C07264=1105.012,382.396,409.215,-179.501,16.996,151.526
C07265=1105.019,382.643,409.178,-179.498,17.001,151.527
C07266=1105.028,383.057,409.117,-179.494,17.008,151.528
C07267=1105.037,383.470,409.056,-179.490,17.016,151.529
C07268=1105.047,383.884,408.995,-179.484,17.024,151.530
C07269=1105.056,384.298,408.934,-179.480,17.032,151.531
C07270=1105.061,384.545,408.897,-179.478,17.037,151.532
C07271=1105.067,384.792,408.860,-179.476,17.041,151.532
C07272=1105.073,385.040,408.823,-179.473,17.046,151.533
C07273=1105.078,385.286,408.787,-179.470,17.051,151.534
C07274=1105.084,385.533,408.750,-179.468,17.056,151.534
C07275=1105.090,385.781,408.713,-179.465,17.060,151.535
C07276=1105.096,386.028,408.677,-179.462,17.065,151.536
C07277=1105.101,386.274,408.640,-179.460,17.070,151.536
C07278=1105.106,386.522,408.603,-179.457,17.075,151.537
C07279=1105.112,386.769,408.566,-179.454,17.080,151.538
C07280=1105.118,387.016,408.529,-179.453,17.084,151.538
C07281=1105.124,387.264,408.492,-179.450,17.089,151.539
C07282=1105.129,387.510,408.456,-179.447,17.094,151.540
C07283=1105.135,387.758,408.419,-179.445,17.098,151.540
C07284=1105.141,388.005,408.382,-179.442,17.104,151.541
C07285=1105.147,388.251,408.344,-179.440,17.108,151.542
C07286=1105.152,388.499,408.307,-179.437,17.113,151.543
C07287=1105.158,388.746,408.270,-179.435,17.118,151.543
C07288=1105.163,388.993,408.234,-179.432,17.123,151.544
C07289=1105.169,389.240,408.197,-179.429,17.128,151.545
C07290=1105.175,389.487,408.160,-179.427,17.133,151.546
C07291=1105.181,389.734,408.122,-179.424,17.138,151.546
C07292=1105.186,389.981,408.085,-179.422,17.143,151.547
C07293=1105.192,390.229,408.048,-179.419,17.148,151.548
C07294=1105.198,390.476,408.012,-179.417,17.153,151.548
C07295=1105.204,390.722,407.974,-179.414,17.158,151.549
C07296=1105.210,390.970,407.937,-179.412,17.164,151.550
C07297=1105.216,391.217,407.900,-179.409,17.168,151.551
C07298=1105.221,391.463,407.863,-179.407,17.174,151.552
C07299=1105.226,391.711,407.826,-179.404,17.179,151.552
C07300=1105.232,391.958,407.789,-179.402,17.184,151.553
C07301=1105.238,392.205,407.751,-179.399,17.189,151.554
C07302=1105.244,392.452,407.714,-179.397,17.194,151.555
C07303=1105.249,392.699,407.676,-179.394,17.199,151.555
C07304=1105.255,392.946,407.639,-179.392,17.204,151.556
C07305=1105.261,393.194,407.602,-179.390,17.210,151.557
C07306=1105.267,393.440,407.564,-179.387,17.215,151.558
C07307=1105.272,393.688,407.527,-179.385,17.220,151.559
C07308=1105.278,393.934,407.489,-179.383,17.225,151.560
C07309=1105.284,394.182,407.452,-179.380,17.231,151.560
C07310=1105.290,394.428,407.415,-179.378,17.236,151.561
C07311=1105.295,394.676,407.378,-179.376,17.241,151.562
C07312=1105.301,394.923,407.340,-179.373,17.247,151.563
C07313=1105.307,395.170,407.303,-179.371,17.252,151.564
C07314=1105.313,395.417,407.265,-179.369,17.257,151.565
C07315=1105.318,395.664,407.228,-179.366,17.263,151.566
C07316=1105.323,395.911,407.190,-179.364,17.268,151.567
C07317=1105.329,396.158,407.152,-179.361,17.274,151.567
C07318=1105.334,396.371,407.119,-179.359,17.278,151.568
C07319=1105.339,396.584,407.087,-179.358,17.283,151.569
C07320=1105.344,396.797,407.055,-179.355,17.288,151.570
C07321=1105.349,397.009,407.023,-179.354,17.293,151.571
C07322=1105.354,397.223,406.990,-179.351,17.298,151.571
C07323=1105.359,397.435,406.958,-179.350,17.302,151.572
C07324=1105.364,397.648,406.925,-179.348,17.307,151.573
C07325=1105.369,397.861,406.892,-179.345,17.312,151.574
C07326=1105.375,398.108,406.855,-179.343,17.317,151.575
C07327=1105.380,398.355,406.818,-179.341,17.323,151.576
C07328=1105.385,398.602,406.779,-179.339,17.328,151.577
C07329=1105.391,398.849,406.741,-179.337,17.334,151.578
C07330=1105.397,399.096,406.704,-179.334,17.340,151.579
C07331=1105.403,399.344,406.666,-179.332,17.346,151.580
C07332=1105.408,399.591,406.628,-179.329,17.351,151.580
C07333=1105.414,399.838,406.590,-179.327,17.357,151.581
C07334=1105.420,400.085,406.552,-179.325,17.363,151.582
C07335=1105.425,400.331,406.514,-179.322,17.369,151.584
C07336=1105.431,400.578,406.476,-179.320,17.375,151.585
C07337=1105.436,400.825,406.438,-179.318,17.380,151.585
C07338=1105.442,401.072,406.400,-179.316,17.386,151.587
C07339=1105.448,401.320,406.362,-179.313,17.392,151.588
C07340=1105.454,401.567,406.324,-179.311,17.398,151.589
C07341=1105.460,401.814,406.287,-179.309,17.404,151.590
C07342=1105.465,402.061,406.248,-179.307,17.409,151.591
C07343=1105.471,402.308,406.211,-179.305,17.416,151.592
C07344=1105.476,402.555,406.172,-179.302,17.422,151.593
C07345=1105.482,402.802,406.134,-179.300,17.428,151.594
C07346=1105.488,403.049,406.096,-179.299,17.434,151.595
C07347=1105.493,403.296,406.058,-179.296,17.440,151.596
C07348=1105.499,403.542,406.019,-179.294,17.446,151.597
C07349=1105.505,403.790,405.981,-179.292,17.452,151.598
C07350=1105.511,404.037,405.942,-179.289,17.458,151.599
C07351=1105.517,404.284,405.905,-179.287,17.464,151.600
C07352=1105.522,404.531,405.866,-179.285,17.470,151.601
C07353=1105.528,404.778,405.828,-179.283,17.476,151.603
C07354=1105.533,405.025,405.790,-179.281,17.482,151.604
C07355=1105.539,405.272,405.752,-179.279,17.488,151.605
C07356=1105.545,405.518,405.713,-179.276,17.495,151.606
C07357=1105.551,405.766,405.675,-179.274,17.501,151.607
C07358=1105.556,406.013,405.637,-179.272,17.508,151.608
C07359=1105.562,406.260,405.598,-179.270,17.514,151.609
C07360=1105.568,406.506,405.560,-179.268,17.520,151.611
C07361=1105.574,406.754,405.521,-179.266,17.527,151.612
C07362=1105.579,407.001,405.483,-179.264,17.532,151.613
C07363=1105.585,407.247,405.444,-179.261,17.539,151.614
C07364=1105.591,407.495,405.406,-179.259,17.545,151.615
C07365=1105.596,407.742,405.367,-179.258,17.552,151.617
C07366=1105.602,407.988,405.329,-179.255,17.558,151.618
C07367=1105.607,408.235,405.290,-179.254,17.565,151.619
C07368=1105.613,408.483,405.252,-179.251,17.572,151.620
C07369=1105.618,408.729,405.213,-179.249,17.578,151.621
C07370=1105.624,408.976,405.174,-179.247,17.584,151.623
C07371=1105.630,409.223,405.135,-179.245,17.591,151.624
C07372=1105.636,409.470,405.097,-179.243,17.598,151.625
C07373=1105.641,409.716,405.058,-179.241,17.604,151.626
C07374=1105.646,409.930,405.025,-179.239,17.610,151.628
C07375=1105.650,410.142,404.992,-179.237,17.616,151.629
C07376=1105.656,410.355,404.958,-179.235,17.622,151.630
C07377=1105.661,410.568,404.924,-179.234,17.627,151.631
C07378=1105.665,410.780,404.891,-179.232,17.633,151.632
C07379=1105.670,410.994,404.857,-179.230,17.639,151.633
C07380=1105.675,411.206,404.824,-179.229,17.645,151.634
C07381=1105.680,411.419,404.791,-179.227,17.651,151.635
C07382=1105.686,411.665,404.752,-179.225,17.657,151.637
C07383=1105.692,411.913,404.713,-179.223,17.664,151.638
C07384=1105.697,412.159,404.674,-179.221,17.671,151.639
C07385=1105.703,412.406,404.635,-179.219,17.678,151.641
C07386=1105.709,412.653,404.596,-179.217,17.685,151.642
C07387=1105.714,412.900,404.557,-179.215,17.692,151.643
C07388=1105.720,413.147,404.518,-179.213,17.699,151.645
C07389=1105.725,413.394,404.480,-179.210,17.706,151.646
C07390=1105.731,413.641,404.440,-179.209,17.713,151.647
C07391=1105.737,413.888,404.401,-179.207,17.720,151.649
C07392=1105.742,414.134,404.362,-179.205,17.726,151.650
C07393=1105.748,414.381,404.323,-179.203,17.734,151.652
C07394=1105.754,414.628,404.285,-179.201,17.741,151.653
C07395=1105.760,414.875,404.245,-179.199,17.748,151.654
C07396=1105.766,415.121,404.206,-179.197,17.755,151.656
C07397=1105.772,415.369,404.167,-179.195,17.762,151.657
C07398=1105.777,415.615,404.128,-179.193,17.770,151.659
C07399=1105.783,415.862,404.088,-179.192,17.776,151.660
C07400=1105.789,416.109,404.049,-179.189,17.784,151.662
C07401=1105.795,416.356,404.010,-179.187,17.791,151.663
C07402=1105.800,416.602,403.971,-179.185,17.799,151.665
C07403=1105.806,416.850,403.931,-179.184,17.805,151.666
C07404=1105.811,417.096,403.892,-179.182,17.813,151.667
C07405=1105.817,417.343,403.852,-179.180,17.820,151.669
C07406=1105.823,417.590,403.813,-179.178,17.828,151.671
C07407=1105.829,417.837,403.774,-179.176,17.835,151.672
C07408=1105.834,418.083,403.735,-179.175,17.843,151.674
C07409=1105.840,418.331,403.695,-179.173,17.850,151.675
C07410=1105.845,418.577,403.656,-179.171,17.858,151.677
C07411=1105.851,418.824,403.616,-179.169,17.865,151.678
C07412=1105.857,419.071,403.577,-179.167,17.873,151.680
C07413=1105.863,419.318,403.538,-179.165,17.881,151.681
C07414=1105.868,419.564,403.497,-179.164,17.888,151.683
C07415=1105.874,419.811,403.458,-179.162,17.895,151.684
C07416=1105.880,420.058,403.419,-179.160,17.903,151.686
C07417=1105.885,420.305,403.379,-179.158,17.911,151.688
C07418=1105.891,420.551,403.339,-179.156,17.919,151.689
C07419=1105.897,420.798,403.300,-179.154,17.927,151.691
C07420=1105.903,421.045,403.260,-179.152,17.934,151.693
C07421=1105.907,421.292,403.221,-179.151,17.942,151.694
C07422=1105.914,421.538,403.180,-179.149,17.950,151.696
C07423=1105.920,421.785,403.141,-179.147,17.958,151.698
C07424=1105.926,422.031,403.101,-179.146,17.965,151.699
C07425=1105.931,422.279,403.061,-179.144,17.973,151.701
C07426=1105.937,422.526,403.022,-179.143,17.982,151.703
C07427=1105.943,422.772,402.982,-179.141,17.989,151.704
C07428=1105.948,423.019,402.942,-179.139,17.997,151.706
C07429=1105.954,423.265,402.902,-179.137,18.005,151.708
C07430=1105.958,423.484,402.867,-179.135,18.013,151.709
C07431=1105.964,423.704,402.832,-179.134,18.020,151.711
C07432=1105.969,423.923,402.795,-179.133,18.027,151.712
C07433=1105.974,424.143,402.760,-179.131,18.035,151.714
C07434=1105.979,424.362,402.725,-179.130,18.042,151.715
C07435=1105.984,424.581,402.689,-179.128,18.050,151.717
C07436=1105.989,424.800,402.654,-179.127,18.057,151.719
C07437=1105.994,425.020,402.619,-179.126,18.064,151.720
C07438=1106.000,425.267,402.578,-179.124,18.072,151.722
C07439=1106.005,425.512,402.538,-179.122,18.080,151.724
C07440=1106.011,425.760,402.498,-179.121,18.088,151.725
C07441=1106.017,426.006,402.458,-179.119,18.098,151.727
C07442=1106.022,426.252,402.418,-179.117,18.106,151.729
C07443=1106.028,426.500,402.378,-179.115,18.114,151.731
C07444=1106.034,426.746,402.337,-179.114,18.123,151.733
C07445=1106.040,426.993,402.297,-179.112,18.131,151.735
C07446=1106.045,427.239,402.257,-179.111,18.139,151.737
C07447=1106.051,427.486,402.217,-179.110,18.148,151.738
C07448=1106.057,427.733,402.177,-179.108,18.156,151.740
C07449=1106.062,427.979,402.136,-179.106,18.165,151.742
C07450=1106.068,428.226,402.096,-179.104,18.174,151.744
C07451=1106.074,428.472,402.056,-179.103,18.183,151.746
C07452=1106.079,428.720,402.015,-179.102,18.191,151.748
C07453=1106.085,428.966,401.976,-179.100,18.200,151.750
C07454=1106.091,429.213,401.935,-179.099,18.209,151.752
C07455=1106.097,429.459,401.894,-179.097,18.218,151.754
C07456=1106.103,429.706,401.854,-179.096,18.226,151.756
C07457=1106.108,429.952,401.814,-179.094,18.235,151.758
C07458=1106.114,430.199,401.773,-179.093,18.244,151.760
C07459=1106.120,430.445,401.733,-179.091,18.254,151.762
C07460=1106.125,430.691,401.692,-179.090,18.262,151.764
C07461=1106.131,430.938,401.652,-179.089,18.271,151.766
C07462=1106.136,431.185,401.611,-179.088,18.280,151.768
C07463=1106.142,431.432,401.570,-179.086,18.290,151.770
C07464=1106.148,431.678,401.530,-179.084,18.298,151.772
C07465=1106.153,431.925,401.490,-179.083,18.308,151.774
C07466=1106.159,432.171,401.449,-179.081,18.317,151.776
C07467=1106.165,432.418,401.407,-179.080,18.326,151.778
C07468=1106.171,432.664,401.367,-179.079,18.335,151.780
C07469=1106.177,432.911,401.327,-179.077,18.345,151.782
C07470=1106.182,433.157,401.286,-179.076,18.354,151.784
C07471=1106.188,433.404,401.245,-179.075,18.363,151.787
C07472=1106.194,433.650,401.204,-179.073,18.373,151.789
C07473=1106.199,433.897,401.163,-179.072,18.382,151.791
C07474=1106.205,434.144,401.123,-179.071,18.391,151.793
C07475=1106.210,434.390,401.082,-179.070,18.401,151.795
C07476=1106.216,434.636,401.041,-179.069,18.410,151.797
C07477=1106.222,434.883,401.000,-179.067,18.421,151.800
C07478=1106.227,435.130,400.959,-179.066,18.430,151.802
C07479=1106.233,435.376,400.918,-179.065,18.439,151.804
C07480=1106.238,435.622,400.877,-179.064,18.449,151.806
C07481=1106.244,435.868,400.836,-179.063,18.459,151.809
C07482=1106.250,436.115,400.795,-179.061,18.469,151.811
C07483=1106.255,436.362,400.754,-179.060,18.478,151.813
C07484=1106.261,436.608,400.713,-179.059,18.488,151.815
C07485=1106.267,436.855,400.672,-179.058,18.498,151.818
C07486=1106.272,437.072,400.636,-179.057,18.507,151.820
C07487=1106.277,437.290,400.600,-179.056,18.516,151.822
C07488=1106.282,437.508,400.563,-179.055,18.524,151.824
C07489=1106.287,437.726,400.526,-179.054,18.533,151.826
C07490=1106.292,437.944,400.490,-179.053,18.542,151.828
C07491=1106.297,438.162,400.454,-179.052,18.551,151.830
C07492=1106.302,438.380,400.418,-179.051,18.560,151.832
C07493=1106.307,438.598,400.381,-179.050,18.569,151.834
C07494=1106.313,438.844,400.340,-179.049,18.579,151.837
C07495=1106.318,439.091,400.299,-179.048,18.589,151.839
C07496=1106.324,439.337,400.257,-179.047,18.600,151.842
C07497=1106.330,439.583,400.216,-179.046,18.609,151.844
C07498=1106.336,439.829,400.175,-179.045,18.620,151.846
C07499=1106.341,440.076,400.133,-179.044,18.630,151.849
C07500=1106.347,440.323,400.092,-179.043,18.641,151.851
C07501=1106.353,440.569,400.050,-179.041,18.651,151.854
C07502=1106.359,440.815,400.009,-179.041,18.661,151.856
C07503=1106.365,441.062,399.968,-179.040,18.672,151.859
C07504=1106.370,441.308,399.926,-179.039,18.682,151.861
C07505=1106.376,441.555,399.885,-179.038,18.693,151.864
C07506=1106.382,441.801,399.843,-179.037,18.704,151.866
C07507=1106.388,442.047,399.802,-179.037,18.714,151.869
C07508=1106.393,442.293,399.760,-179.036,18.725,151.872
C07509=1106.399,442.540,399.718,-179.034,18.736,151.874
C07510=1106.405,442.786,399.677,-179.034,18.747,151.877
C07511=1106.410,443.032,399.635,-179.033,18.758,151.879
C07512=1106.416,443.279,399.593,-179.032,18.769,151.882
C07513=1106.421,443.525,399.551,-179.032,18.779,151.885
C07514=1106.427,443.771,399.510,-179.031,18.790,151.887
C07515=1106.433,444.018,399.468,-179.030,18.801,151.890
C07516=1106.438,444.264,399.426,-179.030,18.812,151.893
C07517=1106.444,444.510,399.385,-179.029,18.823,151.895
C07518=1106.449,444.757,399.343,-179.029,18.834,151.898
C07519=1106.455,445.003,399.301,-179.029,18.845,151.901
C07520=1106.461,445.249,399.259,-179.030,18.855,151.904
C07521=1106.467,445.496,399.218,-179.030,18.866,151.907
C07522=1106.472,445.742,399.176,-179.030,18.877,151.909
C07523=1106.478,445.988,399.134,-179.031,18.887,151.912
C07524=1106.483,446.234,399.091,-179.032,18.898,151.915
C07525=1106.489,446.480,399.050,-179.032,18.909,151.918
C07526=1106.494,446.727,399.008,-179.033,18.920,151.921
C07527=1106.501,446.974,398.966,-179.034,18.930,151.924
C07528=1106.506,447.220,398.924,-179.035,18.941,151.927
C07529=1106.512,447.467,398.883,-179.036,18.952,151.930
C07530=1106.518,447.713,398.840,-179.037,18.963,151.933
C07531=1106.523,447.959,398.798,-179.039,18.973,151.936
C07532=1106.529,448.205,398.756,-179.040,18.984,151.939
C07533=1106.534,448.452,398.714,-179.042,18.994,151.942
C07534=1106.539,448.698,398.671,-179.043,19.005,151.945
C07535=1106.546,448.945,398.630,-179.045,19.015,151.948
C07536=1106.551,449.191,398.588,-179.047,19.026,151.951
C07537=1106.558,449.437,398.545,-179.049,19.037,151.954
C07538=1106.563,449.683,398.503,-179.050,19.047,151.957
C07539=1106.568,449.930,398.461,-179.053,19.058,151.960
C07540=1106.574,450.175,398.419,-179.054,19.068,151.963
C07541=1106.579,450.422,398.377,-179.057,19.079,151.966
C07542=1106.174,450.414,398.257,-179.136,19.309,152.039
C07543=1106.168,450.169,398.299,-179.134,19.299,152.036
C07544=1106.162,449.922,398.341,-179.132,19.288,152.033
C07545=1106.157,449.676,398.384,-179.130,19.277,152.030
C07546=1106.151,449.430,398.425,-179.128,19.267,152.027
C07547=1106.145,449.183,398.468,-179.126,19.256,152.024
C07548=1106.140,448.937,398.510,-179.125,19.245,152.021
C07549=1106.134,448.691,398.552,-179.123,19.235,152.018
C07550=1106.129,448.444,398.594,-179.121,19.224,152.015
C07551=1106.123,448.198,398.637,-179.120,19.213,152.012
C07552=1106.116,447.952,398.678,-179.118,19.203,152.009
C07553=1106.111,447.705,398.720,-179.117,19.192,152.006
C07554=1106.105,447.459,398.763,-179.116,19.181,152.003
C07555=1106.100,447.213,398.805,-179.115,19.170,152.000
C07556=1106.095,446.966,398.847,-179.114,19.160,151.997
C07557=1106.089,446.720,398.888,-179.113,19.149,151.994
C07558=1106.083,446.474,398.931,-179.112,19.138,151.991
C07559=1106.077,446.228,398.972,-179.112,19.127,151.988
C07560=1106.071,445.981,399.015,-179.112,19.116,151.986
C07561=1106.066,445.734,399.057,-179.111,19.106,151.983
C07562=1106.060,445.489,399.099,-179.111,19.095,151.980
C07563=1106.055,445.242,399.141,-179.110,19.084,151.977
C07564=1106.049,444.996,399.183,-179.110,19.073,151.974
C07565=1106.043,444.750,399.224,-179.110,19.062,151.971
C07566=1106.038,444.503,399.266,-179.110,19.051,151.969
C07567=1106.032,444.257,399.308,-179.110,19.040,151.966
C07568=1106.026,444.011,399.350,-179.111,19.029,151.963
C07569=1106.020,443.765,399.392,-179.112,19.018,151.960
C07570=1106.015,443.519,399.434,-179.112,19.008,151.958
C07571=1106.009,443.272,399.475,-179.113,18.996,151.955
C07572=1106.004,443.026,399.517,-179.114,18.985,151.952
C07573=1105.998,442.780,399.559,-179.115,18.974,151.950
C07574=1105.992,442.533,399.600,-179.115,18.964,151.947
C07575=1105.987,442.287,399.642,-179.117,18.953,151.945
C07576=1105.980,442.040,399.684,-179.118,18.942,151.942
C07577=1105.975,441.795,399.725,-179.118,18.931,151.939
C07578=1105.969,441.548,399.767,-179.119,18.920,151.937
C07579=1105.964,441.301,399.808,-179.121,18.909,151.934
C07580=1105.958,441.055,399.849,-179.121,18.899,151.932
C07581=1105.952,440.809,399.891,-179.122,18.888,151.929
C07582=1105.947,440.562,399.933,-179.123,18.878,151.927
C07583=1105.941,440.316,399.974,-179.124,18.867,151.924
C07584=1105.935,440.070,400.016,-179.126,18.857,151.922
C07585=1105.929,439.824,400.057,-179.126,18.847,151.919
C07586=1105.923,439.577,400.098,-179.127,18.836,151.917
C07587=1105.917,439.331,400.140,-179.128,18.826,151.914
C07588=1105.912,439.084,400.182,-179.130,18.815,151.912
C07589=1105.906,438.838,400.223,-179.131,18.805,151.910
C07590=1105.901,438.591,400.264,-179.132,18.795,151.907
C07591=1105.896,438.375,400.300,-179.133,18.786,151.905
C07592=1105.890,438.159,400.336,-179.134,18.777,151.903
C07593=1105.885,437.943,400.373,-179.135,18.768,151.901
C07594=1105.880,437.727,400.409,-179.136,18.759,151.899
C07595=1105.875,437.512,400.444,-179.137,18.750,151.897
C07596=1105.870,437.297,400.480,-179.138,18.742,151.895
C07597=1105.865,437.081,400.517,-179.139,18.733,151.893
C07598=1105.860,436.865,400.553,-179.140,18.724,151.891
C07599=1105.854,436.618,400.594,-179.141,18.714,151.888
C07600=1105.848,436.372,400.635,-179.143,18.704,151.886
C07601=1105.843,436.126,400.675,-179.143,18.695,151.884
C07602=1105.837,435.879,400.717,-179.145,18.684,151.881
C07603=1105.832,435.633,400.758,-179.146,18.675,151.879
C07604=1105.826,435.386,400.799,-179.148,18.665,151.877
C07605=1105.820,435.140,400.840,-179.149,18.655,151.875
C07606=1105.814,434.893,400.881,-179.150,18.646,151.872
C07607=1105.809,434.647,400.922,-179.151,18.636,151.870
C07608=1105.804,434.400,400.962,-179.152,18.626,151.868
C07609=1105.798,434.154,401.004,-179.154,18.616,151.866
C07610=1105.792,433.907,401.045,-179.155,18.607,151.864
C07611=1105.786,433.661,401.085,-179.157,18.597,151.861
C07612=1105.780,433.414,401.127,-179.158,18.588,151.859
C07613=1105.775,433.168,401.167,-179.159,18.579,151.857
C07614=1105.770,432.921,401.208,-179.161,18.569,151.855
C07615=1105.764,432.675,401.249,-179.162,18.560,151.853
C07616=1105.758,432.428,401.290,-179.163,18.550,151.851
C07617=1105.752,432.182,401.330,-179.165,18.541,151.849
C07618=1105.747,431.936,401.371,-179.166,18.532,151.847
C07619=1105.741,431.689,401.411,-179.167,18.523,151.845
C07620=1105.735,431.442,401.452,-179.169,18.513,151.842
C07621=1105.730,431.195,401.493,-179.171,18.504,151.840
C07622=1105.723,430.949,401.534,-179.172,18.495,151.838
C07623=1105.718,430.703,401.574,-179.173,18.486,151.836
C07624=1105.712,430.456,401.615,-179.175,18.477,151.834
C07625=1105.707,430.210,401.656,-179.176,18.468,151.832
C07626=1105.701,429.963,401.696,-179.178,18.459,151.830
C07627=1105.695,429.717,401.736,-179.179,18.450,151.828
C07628=1105.690,429.470,401.777,-179.181,18.441,151.826
C07629=1105.684,429.223,401.818,-179.182,18.432,151.824
C07630=1105.678,428.977,401.858,-179.183,18.423,151.822
C07631=1105.672,428.730,401.898,-179.185,18.415,151.820
C07632=1105.667,428.484,401.939,-179.187,18.405,151.818
C07633=1105.661,428.237,401.978,-179.189,18.397,151.816
C07634=1105.655,427.990,402.019,-179.190,18.388,151.814
C07635=1105.649,427.743,402.059,-179.191,18.380,151.813
C07636=1105.644,427.497,402.100,-179.193,18.371,151.811
C07637=1105.638,427.250,402.140,-179.195,18.363,151.809
C07638=1105.632,427.004,402.180,-179.197,18.353,151.807
C07639=1105.627,426.757,402.220,-179.198,18.345,151.805
C07640=1105.621,426.511,402.260,-179.200,18.336,151.803
C07641=1105.615,426.264,402.301,-179.201,18.328,151.801
C07642=1105.609,426.017,402.341,-179.203,18.319,151.800
C07643=1105.604,425.771,402.381,-179.204,18.311,151.798
C07644=1105.598,425.524,402.422,-179.206,18.303,151.796
C07645=1105.592,425.277,402.462,-179.207,18.294,151.794
C07646=1105.587,425.031,402.501,-179.209,18.286,151.792
C07647=1105.581,424.811,402.537,-179.211,18.278,151.791
C07648=1105.576,424.592,402.573,-179.212,18.271,151.789
C07649=1105.572,424.372,402.608,-179.214,18.264,151.788
C07650=1105.567,424.153,402.644,-179.215,18.256,151.786
C07651=1105.561,423.933,402.679,-179.216,18.249,151.784
C07652=1105.556,423.714,402.715,-179.219,18.241,151.783
C07653=1105.552,423.494,402.750,-179.220,18.234,151.781
C07654=1105.547,423.275,402.786,-179.222,18.227,151.780
C07655=1105.541,423.028,402.826,-179.224,18.219,151.778
C07656=1105.534,422.782,402.866,-179.225,18.211,151.776
C07657=1105.530,422.535,402.906,-179.227,18.202,151.775
C07658=1105.523,422.288,402.946,-179.229,18.194,151.773
C07659=1105.517,422.041,402.985,-179.230,18.187,151.771
C07660=1105.512,421.795,403.025,-179.232,18.179,151.770
C07661=1105.506,421.548,403.065,-179.233,18.171,151.768
C07662=1105.500,421.301,403.105,-179.235,18.163,151.766
C07663=1105.495,421.054,403.144,-179.237,18.155,151.765
C07664=1105.489,420.808,403.184,-179.239,18.147,151.763
C07665=1105.483,420.561,403.223,-179.241,18.140,151.761
C07666=1105.477,420.314,403.263,-179.243,18.132,151.760
C07667=1105.472,420.067,403.304,-179.245,18.124,151.758
C07668=1105.466,419.821,403.343,-179.247,18.116,151.756
C07669=1105.460,419.574,403.382,-179.248,18.108,151.755
C07670=1105.455,419.327,403.421,-179.250,18.100,151.753
C07671=1105.449,419.080,403.462,-179.252,18.093,151.752
C07672=1105.444,418.834,403.501,-179.254,18.086,151.750
C07673=1105.438,418.587,403.540,-179.256,18.078,151.749
C07674=1105.432,418.340,403.579,-179.258,18.070,151.747
C07675=1105.427,418.093,403.619,-179.260,18.062,151.745
C07676=1105.421,417.847,403.659,-179.262,18.055,151.744
C07677=1105.415,417.599,403.698,-179.263,18.047,151.742
C07678=1105.409,417.354,403.738,-179.265,18.040,151.741
C07679=1105.403,417.106,403.777,-179.267,18.033,151.739
C07680=1105.399,416.860,403.817,-179.269,18.025,151.738
C07681=1105.392,416.613,403.856,-179.271,18.017,151.736
C07682=1105.387,416.366,403.895,-179.273,18.010,151.735
C07683=1105.381,416.119,403.935,-179.275,18.003,151.733
C07684=1105.375,415.872,403.974,-179.277,17.996,151.732
C07685=1105.369,415.625,404.013,-179.279,17.988,151.730
C07686=1105.363,415.378,404.053,-179.281,17.981,151.729
C07687=1105.358,415.131,404.091,-179.282,17.974,151.728
C07688=1105.352,414.884,404.130,-179.285,17.967,151.726
C07689=1105.347,414.638,404.170,-179.287,17.960,151.725
C07690=1105.341,414.391,404.209,-179.288,17.953,151.723
C07691=1105.335,414.144,404.248,-179.291,17.946,151.722
C07692=1105.330,413.898,404.287,-179.293,17.938,151.720
C07693=1105.324,413.651,404.327,-179.294,17.932,151.719
C07694=1105.318,413.403,404.365,-179.296,17.924,151.718
C07695=1105.312,413.157,404.404,-179.299,17.917,151.716
C07696=1105.306,412.910,404.443,-179.300,17.910,151.715
C07697=1105.300,412.663,404.482,-179.303,17.903,151.714
C07698=1105.295,412.416,404.521,-179.305,17.896,151.712
C07699=1105.289,412.169,404.560,-179.306,17.889,151.711
C07700=1105.283,411.922,404.599,-179.309,17.882,151.709
C07701=1105.278,411.675,404.637,-179.311,17.875,151.708
C07702=1105.272,411.428,404.677,-179.313,17.869,151.707
C07703=1105.267,411.215,404.710,-179.314,17.862,151.706
C07704=1105.262,411.003,404.744,-179.316,17.857,151.704
C07705=1105.257,410.790,404.777,-179.318,17.851,151.703
C07706=1105.252,410.577,404.811,-179.319,17.845,151.702
C07707=1105.248,410.365,404.845,-179.321,17.839,151.701
C07708=1105.243,410.151,404.877,-179.323,17.833,151.700
C07709=1105.238,409.938,404.911,-179.325,17.828,151.699
C07710=1105.233,409.725,404.945,-179.327,17.821,151.698
C07711=1105.227,409.479,404.984,-179.329,17.815,151.696
C07712=1105.222,409.232,405.022,-179.331,17.808,151.695
C07713=1105.216,408.984,405.061,-179.333,17.802,151.694
C07714=1105.210,408.738,405.099,-179.335,17.795,151.693
C07715=1105.205,408.491,405.138,-179.337,17.788,151.691
C07716=1105.199,408.244,405.177,-179.339,17.781,151.690
C07717=1105.194,407.996,405.215,-179.341,17.776,151.689
C07718=1105.187,407.750,405.254,-179.344,17.769,151.688
C07719=1105.182,407.503,405.292,-179.346,17.762,151.686
C07720=1105.177,407.256,405.331,-179.348,17.755,151.685
C07721=1105.170,407.009,405.369,-179.350,17.749,151.684
C07722=1105.165,406.762,405.408,-179.352,17.743,151.683
C07723=1105.159,406.515,405.447,-179.354,17.737,151.682
C07724=1105.154,406.268,405.486,-179.356,17.730,151.680
C07725=1105.148,406.021,405.523,-179.359,17.724,151.679
C07726=1105.142,405.774,405.562,-179.360,17.717,151.678
C07727=1105.136,405.527,405.600,-179.362,17.711,151.677
C07728=1105.131,405.280,405.639,-179.365,17.705,151.676
C07729=1105.126,405.033,405.677,-179.367,17.699,151.675
C07730=1105.119,404.786,405.715,-179.369,17.692,151.674
C07731=1105.114,404.539,405.754,-179.371,17.686,151.672
C07732=1105.108,404.292,405.791,-179.373,17.680,151.671
C07733=1105.103,404.046,405.831,-179.376,17.674,151.670
C07734=1105.096,403.798,405.869,-179.378,17.668,151.669
C07735=1105.091,403.551,405.907,-179.380,17.662,151.668
C07736=1105.085,403.305,405.945,-179.383,17.655,151.667
C07737=1105.080,403.057,405.983,-179.385,17.650,151.666
C07738=1105.073,402.810,406.021,-179.387,17.644,151.665
C07739=1105.068,402.563,406.060,-179.389,17.637,151.664
C07740=1105.062,402.316,406.097,-179.391,17.631,151.663
C07741=1105.057,402.069,406.136,-179.393,17.625,151.661
C07742=1105.051,401.822,406.173,-179.395,17.620,151.661
C07743=1105.045,401.575,406.212,-179.398,17.613,151.659
C07744=1105.040,401.328,406.250,-179.400,17.608,151.658
C07745=1105.034,401.081,406.288,-179.402,17.602,151.657
C07746=1105.029,400.834,406.326,-179.404,17.596,151.656
C07747=1105.023,400.587,406.364,-179.407,17.589,151.655
C07748=1105.017,400.340,406.402,-179.409,17.584,151.654
C07749=1105.011,400.093,406.440,-179.411,17.578,151.653
C07750=1105.005,399.846,406.478,-179.414,17.572,151.652
C07751=1105.000,399.599,406.516,-179.416,17.566,151.651
C07752=1104.994,399.352,406.553,-179.418,17.560,151.650
C07753=1104.988,399.105,406.591,-179.421,17.555,151.649
C07754=1104.983,398.858,406.629,-179.423,17.549,151.648
C07755=1104.977,398.611,406.667,-179.425,17.544,151.647
C07756=1104.971,398.364,406.705,-179.428,17.537,151.646
C07757=1104.965,398.116,406.742,-179.430,17.532,151.645
C07758=1104.960,397.869,406.781,-179.432,17.526,151.644
C07759=1104.955,397.657,406.813,-179.434,17.522,151.644
C07760=1104.950,397.443,406.846,-179.436,17.516,151.643
C07761=1104.945,397.231,406.879,-179.438,17.512,151.642
C07762=1104.940,397.017,406.911,-179.440,17.507,151.641
C07763=1104.936,396.805,406.944,-179.442,17.502,151.640
C07764=1104.931,396.591,406.976,-179.445,17.497,151.639
C07765=1104.925,396.379,407.008,-179.446,17.492,151.639
C07766=1104.921,396.166,407.040,-179.448,17.488,151.638
C07767=1104.915,395.919,407.079,-179.451,17.482,151.637
C07768=1104.910,395.672,407.116,-179.453,17.477,151.636
C07769=1104.903,395.424,407.154,-179.455,17.471,151.635
C07770=1104.898,395.177,407.191,-179.458,17.466,151.634
C07771=1104.892,394.930,407.229,-179.460,17.460,151.633
C07772=1104.886,394.683,407.266,-179.463,17.455,151.633
C07773=1104.880,394.436,407.303,-179.465,17.450,151.632
C07774=1104.874,394.189,407.341,-179.467,17.444,151.631
C07775=1104.869,393.942,407.378,-179.469,17.439,151.630
C07776=1104.864,393.695,407.416,-179.472,17.434,151.629
C07777=1104.858,393.447,407.453,-179.474,17.428,151.628
C07778=1104.852,393.201,407.491,-179.476,17.423,151.627
C07779=1104.847,392.953,407.528,-179.479,17.418,151.627
C07780=1104.841,392.706,407.565,-179.481,17.413,151.626
C07781=1104.836,392.460,407.603,-179.485,17.407,151.625
C07782=1104.830,392.213,407.640,-179.487,17.402,151.624
C07783=1104.824,391.966,407.678,-179.490,17.396,151.623
C07784=1104.819,391.718,407.715,-179.492,17.391,151.623
C07785=1104.812,391.471,407.751,-179.494,17.386,151.622
C07786=1104.806,391.225,407.789,-179.497,17.381,151.621
C07787=1104.801,390.977,407.826,-179.499,17.376,151.620
C07788=1104.795,390.730,407.863,-179.502,17.371,151.619
C07789=1104.789,390.483,407.901,-179.504,17.365,151.619
C07790=1104.784,390.236,407.938,-179.507,17.361,151.618
C07791=1104.778,389.988,407.975,-179.509,17.355,151.617
C07792=1104.772,389.741,408.011,-179.512,17.350,151.616
C07793=1104.766,389.495,408.049,-179.515,17.346,151.616
C07794=1104.760,389.247,408.086,-179.517,17.340,151.615
C07795=1104.755,389.000,408.123,-179.519,17.335,151.614
C07796=1104.750,388.753,408.160,-179.522,17.330,151.613
C07797=1104.744,388.507,408.197,-179.525,17.325,151.613
C07798=1104.737,388.260,408.234,-179.527,17.321,151.612
C07799=1104.732,388.012,408.271,-179.529,17.316,151.611
C07800=1104.726,387.765,408.308,-179.532,17.311,151.610
C07801=1104.721,387.517,408.345,-179.534,17.306,151.610
C07802=1104.715,387.271,408.381,-179.537,17.301,151.609
C07803=1104.709,387.024,408.418,-179.539,17.296,151.608
C07804=1104.704,386.776,408.455,-179.542,17.291,151.608
C07805=1104.698,386.529,408.492,-179.545,17.286,151.607
C07806=1104.691,386.283,408.529,-179.547,17.281,151.606
C07807=1104.686,386.036,408.566,-179.550,17.276,151.605
C07808=1104.681,385.789,408.603,-179.553,17.272,151.605
C07809=1104.675,385.541,408.640,-179.555,17.267,151.604
C07810=1104.669,385.294,408.676,-179.558,17.262,151.603
C07811=1104.664,385.046,408.713,-179.560,17.257,151.603
C07812=1104.659,384.799,408.749,-179.562,17.253,151.602
C07813=1104.652,384.552,408.786,-179.565,17.248,151.601
C07814=1104.647,384.305,408.823,-179.568,17.243,151.601
C07815=1104.637,383.891,408.884,-179.572,17.235,151.600
C07816=1104.629,383.477,408.946,-179.577,17.227,151.599
C07817=1104.619,383.063,409.007,-179.581,17.219,151.598
C07818=1104.609,382.651,409.069,-179.586,17.212,151.597
C07819=1104.603,382.403,409.104,-179.589,17.207,151.596
C07820=1104.598,382.155,409.141,-179.591,17.202,151.595
C07821=1104.591,381.908,409.178,-179.593,17.198,151.595
C07822=1104.586,381.661,409.215,-179.596,17.194,151.594
C07823=1104.580,381.414,409.250,-179.599,17.189,151.594
C07824=1104.575,381.167,409.287,-179.602,17.184,151.593
C07825=1104.568,380.920,409.324,-179.605,17.180,151.592
C07826=1104.564,380.672,409.360,-179.607,17.176,151.592
C07827=1104.557,380.425,409.396,-179.609,17.171,151.591
C07828=1104.551,380.178,409.433,-179.612,17.167,151.591
C07829=1104.546,379.930,409.469,-179.615,17.162,151.590
C07830=1104.540,379.684,409.505,-179.618,17.158,151.590
C07831=1104.534,379.437,409.542,-179.620,17.153,151.589
C07832=1104.528,379.189,409.578,-179.623,17.149,151.589
C07833=1104.523,378.942,409.614,-179.626,17.145,151.588
C07834=1104.517,378.695,409.650,-179.629,17.140,151.587
C07835=1104.511,378.447,409.687,-179.631,17.136,151.587
C07836=1104.506,378.200,409.723,-179.634,17.132,151.586
C07837=1104.500,377.953,409.759,-179.637,17.127,151.586
C07838=1104.495,377.706,409.795,-179.640,17.122,151.585
C07839=1104.489,377.459,409.831,-179.642,17.119,151.585
C07840=1104.483,377.211,409.867,-179.645,17.114,151.584
C07841=1104.478,376.964,409.904,-179.648,17.110,151.584
C07842=1104.472,376.717,409.940,-179.651,17.105,151.583
C07843=1104.466,376.469,409.975,-179.653,17.101,151.583
C07844=1104.461,376.222,410.012,-179.656,17.097,151.582
C07845=1104.455,375.975,410.048,-179.659,17.093,151.582
C07846=1104.449,375.728,410.084,-179.661,17.089,151.581
C07847=1104.444,375.480,410.120,-179.664,17.084,151.581
C07848=1104.438,375.233,410.155,-179.667,17.080,151.580
C07849=1104.432,374.986,410.191,-179.670,17.076,151.580
C07850=1104.427,374.738,410.228,-179.672,17.072,151.579
C07851=1104.421,374.491,410.264,-179.675,17.067,151.579
C07852=1104.415,374.244,410.299,-179.678,17.063,151.578
C07853=1104.410,373.997,410.335,-179.681,17.060,151.578
C07854=1104.404,373.750,410.371,-179.684,17.055,151.578
C07855=1104.398,373.502,410.407,-179.687,17.051,151.577
C07856=1104.393,373.255,410.443,-179.689,17.047,151.577
C07857=1104.387,373.007,410.479,-179.692,17.043,151.576
C07858=1104.381,372.761,410.515,-179.695,17.039,151.576
C07859=1104.375,372.513,410.550,-179.697,17.035,151.575
C07860=1104.370,372.266,410.586,-179.700,17.031,151.575
C07861=1104.364,372.018,410.621,-179.704,17.027,151.575
C07862=1104.358,371.771,410.657,-179.706,17.023,151.574
C07863=1104.353,371.524,410.693,-179.709,17.019,151.574
C07864=1104.347,371.276,410.729,-179.711,17.015,151.573
C07865=1104.341,371.029,410.764,-179.715,17.011,151.573
C07866=1104.335,370.781,410.800,-179.718,17.007,151.573
C07867=1104.327,370.394,410.856,-179.722,17.001,151.572
C07868=1104.317,370.008,410.911,-179.726,16.995,151.571
C07869=1104.309,369.621,410.966,-179.731,16.989,151.571
C07870=1104.300,369.234,411.022,-179.736,16.983,151.570
C07871=1104.294,368.986,411.058,-179.738,16.979,151.570
C07872=1104.289,368.739,411.094,-179.741,16.975,151.569
C07873=1104.283,368.491,411.129,-179.744,16.972,151.569
C07874=1104.277,368.244,411.165,-179.747,16.968,151.569
C07875=1104.271,367.997,411.200,-179.750,16.964,151.568
C07876=1104.266,367.749,411.235,-179.753,16.960,151.568
C07877=1104.260,367.502,411.271,-179.756,16.956,151.568
C07878=1104.255,367.255,411.306,-179.758,16.952,151.567
C07879=1104.249,367.008,411.341,-179.762,16.948,151.567
C07880=1104.243,366.760,411.377,-179.764,16.945,151.567
C07881=1104.238,366.512,411.412,-179.767,16.941,151.566
C07882=1104.232,366.265,411.448,-179.771,16.937,151.566
C07883=1104.226,366.018,411.482,-179.773,16.934,151.566
C07884=1104.220,365.770,411.518,-179.776,16.930,151.565
C07885=1104.215,365.523,411.553,-179.779,16.926,151.565
C07886=1104.209,365.276,411.588,-179.782,16.922,151.565
C07887=1104.203,365.028,411.624,-179.785,16.919,151.564
C07888=1104.198,364.780,411.658,-179.788,16.915,151.564
C07889=1104.192,364.533,411.694,-179.791,16.912,151.564
C07890=1104.186,364.286,411.729,-179.794,16.908,151.564
C07891=1104.181,364.039,411.764,-179.796,16.905,151.563
C07892=1104.175,363.791,411.799,-179.800,16.901,151.563
C07893=1104.170,363.543,411.834,-179.802,16.898,151.563
C07894=1104.163,363.296,411.869,-179.806,16.894,151.562
C07895=1104.158,363.048,411.904,-179.808,16.890,151.562
C07896=1104.152,362.801,411.939,-179.812,16.887,151.562
C07897=1104.147,362.553,411.974,-179.814,16.883,151.562
C07898=1104.141,362.306,412.009,-179.817,16.879,151.561
C07899=1104.135,362.058,412.044,-179.820,16.876,151.561
C07900=1104.129,361.811,412.079,-179.823,16.872,151.561
C07901=1104.124,361.564,412.114,-179.826,16.869,151.561
C07902=1104.118,361.316,412.149,-179.829,16.865,151.560
C07903=1104.112,361.069,412.184,-179.832,16.862,151.560
C07904=1104.107,360.822,412.219,-179.835,16.858,151.560
C07905=1104.101,360.574,412.254,-179.838,16.855,151.560
C07906=1104.095,360.326,412.288,-179.841,16.851,151.559
C07907=1104.090,360.079,412.324,-179.844,16.848,151.559
C07908=1104.084,359.831,412.358,-179.847,16.845,151.559
C07909=1104.078,359.583,412.393,-179.850,16.841,151.559
C07910=1104.072,359.337,412.427,-179.853,16.838,151.558
C07911=1104.067,359.089,412.462,-179.857,16.835,151.558
C07912=1104.061,358.841,412.497,-179.859,16.831,151.558
C07913=1104.055,358.594,412.532,-179.863,16.828,151.558
C07914=1104.050,358.347,412.566,-179.865,16.825,151.558
C07915=1104.044,358.099,412.601,-179.869,16.821,151.558
C07916=1104.039,357.851,412.635,-179.871,16.818,151.557
C07917=1104.032,357.604,412.670,-179.874,16.815,151.557
C07918=1104.027,357.356,412.705,-179.878,16.811,151.557
C07919=1104.018,356.984,412.757,-179.882,16.806,151.557
C07920=1104.010,356.612,412.809,-179.887,16.802,151.556
C07921=1104.001,356.240,412.861,-179.892,16.796,151.556
C07922=1103.992,355.868,412.913,-179.896,16.792,151.556
C07923=1103.987,355.620,412.947,-179.899,16.788,151.556
C07924=1103.981,355.373,412.981,-179.902,16.785,151.555
C07925=1103.976,355.125,413.016,-179.905,16.782,151.555
C07926=1103.970,354.877,413.050,-179.908,16.778,151.555
C07927=1103.965,354.630,413.085,-179.911,16.775,151.555
C07928=1103.959,354.382,413.119,-179.915,16.772,151.555
C07929=1103.953,354.135,413.153,-179.917,16.769,151.555
C07930=1103.948,353.887,413.188,-179.920,16.766,151.555
C07931=1103.941,353.639,413.222,-179.924,16.763,151.554
C07932=1103.936,353.392,413.257,-179.927,16.760,151.554
C07933=1103.930,353.145,413.291,-179.929,16.757,151.554
C07934=1103.924,352.897,413.325,-179.933,16.753,151.554
C07935=1103.919,352.650,413.360,-179.936,16.750,151.554
C07936=1103.913,352.402,413.394,-179.939,16.748,151.554
C07937=1103.907,352.154,413.427,-179.942,16.744,151.554
C07938=1103.902,351.906,413.462,-179.945,16.741,151.553
C07939=1103.896,351.659,413.496,-179.948,16.738,151.553
C07940=1103.891,351.412,413.530,-179.952,16.735,151.553
C07941=1103.885,351.164,413.564,-179.955,16.732,151.553
C07942=1103.879,350.916,413.599,-179.958,16.729,151.553
C07943=1103.873,350.668,413.633,-179.961,16.726,151.553
C07944=1103.868,350.421,413.667,-179.964,16.723,151.553
C07945=1103.862,350.174,413.701,-179.967,16.720,151.553
C07946=1103.857,349.926,413.735,-179.971,16.716,151.553
C07947=1103.851,349.678,413.769,-179.974,16.714,151.553
C07948=1103.845,349.431,413.803,-179.976,16.711,151.552
C07949=1103.839,349.184,413.837,-179.980,16.708,151.552
C07950=1103.834,348.935,413.871,-179.983,16.705,151.552
C07951=1103.828,348.687,413.905,-179.986,16.702,151.552
C07952=1103.822,348.440,413.939,-179.989,16.699,151.552
C07953=1103.817,348.192,413.973,-179.993,16.696,151.552
C07954=1103.811,347.945,414.007,-179.995,16.693,151.552
C07955=1103.805,347.698,414.041,-179.998,16.690,151.552
C07956=1103.800,347.449,414.075,179.998,16.687,151.552
C07957=1103.794,347.202,414.109,179.995,16.684,151.552
C07958=1103.789,346.954,414.142,179.992,16.682,151.552
C07959=1103.783,346.707,414.176,179.989,16.679,151.552
C07960=1103.777,346.459,414.209,179.985,16.675,151.552
C07961=1103.771,346.212,414.243,179.982,16.673,151.552
C07962=1103.766,345.964,414.277,179.979,16.670,151.552
C07963=1103.760,345.717,414.311,179.976,16.667,151.552
C07964=1103.754,345.468,414.345,179.973,16.664,151.552
C07965=1103.749,345.220,414.379,179.970,16.661,151.551
C07966=1103.743,344.972,414.413,179.967,16.659,151.551
C07967=1103.737,344.725,414.447,179.964,16.656,151.551
C07968=1103.731,344.478,414.479,179.960,16.653,151.551
C07969=1103.725,344.230,414.513,179.957,16.650,151.551
C07970=1103.720,343.982,414.547,179.954,16.648,151.551
C07971=1103.711,343.612,414.597,179.949,16.644,151.551
C07972=1103.703,343.242,414.646,179.944,16.639,151.551
C07973=1103.694,342.873,414.697,179.939,16.635,151.551
C07974=1103.686,342.502,414.747,179.935,16.631,151.551
C07975=1103.681,342.254,414.781,179.932,16.629,151.551
C07976=1103.675,342.007,414.815,179.928,16.625,151.551
C07977=1103.668,341.759,414.847,179.925,16.623,151.551
C07978=1103.663,341.512,414.881,179.922,16.620,151.551
C07979=1103.657,341.264,414.914,179.919,16.618,151.551
C07980=1103.652,341.016,414.947,179.916,16.615,151.551
C07981=1103.646,340.768,414.981,179.912,16.612,151.551
C07982=1103.640,340.521,415.015,179.909,16.610,151.551
C07983=1103.635,340.273,415.048,179.905,16.607,151.551
C07984=1103.629,340.025,415.081,179.902,16.605,151.551
C07985=1103.624,339.778,415.114,179.899,16.602,151.551
C07986=1103.618,339.530,415.147,179.896,16.599,151.551
C07987=1103.612,339.282,415.181,179.892,16.596,151.551
C07988=1103.607,339.034,415.214,179.889,16.594,151.551
C07989=1103.601,338.787,415.248,179.886,16.591,151.551
C07990=1103.595,338.539,415.281,179.883,16.589,151.552
C07991=1103.589,338.291,415.314,179.880,16.586,151.552
C07992=1103.584,338.043,415.347,179.877,16.584,151.552
C07993=1103.578,337.796,415.381,179.873,16.581,151.552
C07994=1103.572,337.548,415.413,179.870,16.578,151.552
C07995=1103.566,337.300,415.447,179.867,16.576,151.552
C07996=1103.561,337.053,415.480,179.863,16.574,151.552
C07997=1103.556,336.805,415.513,179.860,16.571,151.552
C07998=1103.550,336.557,415.545,179.857,16.569,151.552
C07999=1103.544,336.309,415.578,179.854,16.566,151.552
C08000=1103.539,336.061,415.612,179.851,16.564,151.552
C08001=1103.532,335.813,415.645,179.847,16.561,151.552
C08002=1103.527,335.565,415.678,179.844,16.558,151.552
C08003=1103.521,335.318,415.711,179.840,16.556,151.552
C08004=1103.516,335.071,415.744,179.837,16.554,151.553
C08005=1103.510,334.823,415.777,179.834,16.551,151.553
C08006=1103.504,334.575,415.809,179.831,16.549,151.553
C08007=1103.498,334.327,415.842,179.828,16.546,151.553
C08008=1103.493,334.079,415.876,179.825,16.544,151.553
C08009=1103.487,333.832,415.908,179.821,16.542,151.553
C08010=1103.482,333.584,415.941,179.818,16.539,151.553
C08011=1103.476,333.335,415.974,179.814,16.536,151.553
C08012=1103.470,333.088,416.007,179.811,16.534,151.553
C08013=1103.465,332.840,416.040,179.808,16.532,151.553
C08014=1103.459,332.592,416.072,179.804,16.529,151.553
C08015=1103.454,332.344,416.105,179.801,16.527,151.553
C08016=1103.447,332.097,416.138,179.798,16.525,151.554
C08017=1103.442,331.848,416.170,179.794,16.522,151.554
C08018=1103.436,331.601,416.203,179.791,16.520,151.554
C08019=1103.430,331.354,416.236,179.788,16.518,151.554
C08020=1103.425,331.105,416.268,179.785,16.516,151.554
C08021=1103.419,330.858,416.301,179.781,16.513,151.554
C08022=1103.413,330.610,416.334,179.778,16.511,151.554
C08023=1103.404,330.234,416.383,179.773,16.508,151.555
C08024=1103.395,329.858,416.433,179.768,16.504,151.555
C08025=1103.387,329.482,416.482,179.763,16.501,151.555
C08026=1103.378,329.106,416.531,179.757,16.497,151.555
C08027=1103.372,328.857,416.564,179.754,16.495,151.555
C08028=1103.366,328.610,416.597,179.751,16.492,151.555
C08029=1103.361,328.362,416.628,179.748,16.490,151.556
C08030=1103.354,328.115,416.661,179.744,16.488,151.556
C08031=1103.349,327.866,416.694,179.741,16.486,151.556
C08032=1103.343,327.618,416.726,179.737,16.484,151.556
C08033=1103.338,327.371,416.758,179.734,16.482,151.556
C08034=1103.332,327.122,416.791,179.731,16.480,151.557
C08035=1103.326,326.875,416.823,179.727,16.477,151.557
C08036=1103.321,326.627,416.855,179.724,16.475,151.557
C08037=1103.315,326.379,416.887,179.721,16.473,151.557
C08038=1103.309,326.131,416.920,179.717,16.471,151.557
C08039=1103.304,325.884,416.952,179.714,16.469,151.557
C08040=1103.298,325.635,416.984,179.711,16.467,151.558
C08041=1103.291,325.388,417.017,179.707,16.464,151.558
C08042=1103.287,325.140,417.049,179.704,16.462,151.558
C08043=1103.281,324.892,417.081,179.700,16.460,151.558
C08044=1103.275,324.644,417.113,179.698,16.459,151.558
C08045=1103.269,324.397,417.146,179.695,16.456,151.558
C08046=1103.263,324.148,417.178,179.691,16.454,151.559
C08047=1103.258,323.901,417.210,179.688,16.452,151.559
C08048=1103.252,323.652,417.242,179.684,16.450,151.559
C08049=1103.246,323.404,417.274,179.681,16.448,151.559
C08050=1103.241,323.157,417.306,179.678,16.446,151.559
C08051=1103.235,322.909,417.338,179.674,16.443,151.559
C08052=1103.229,322.662,417.370,179.671,16.441,151.560
C08053=1103.223,322.413,417.402,179.668,16.439,151.560
C08054=1103.218,322.165,417.435,179.664,16.437,151.560
C08055=1103.213,321.917,417.466,179.661,16.435,151.560
C08056=1103.207,321.669,417.498,179.657,16.433,151.560
C08057=1103.201,321.422,417.530,179.654,16.431,151.561
C08058=1103.195,321.173,417.562,179.651,16.429,151.561
C08059=1103.190,320.926,417.594,179.647,16.427,151.561
C08060=1103.184,320.678,417.626,179.644,16.424,151.561
C08061=1103.179,320.430,417.657,179.640,16.423,151.562
C08062=1103.173,320.182,417.690,179.637,16.421,151.562
C08063=1103.168,319.934,417.722,179.633,16.418,151.562
C08064=1103.162,319.686,417.754,179.631,16.417,151.562
C08065=1103.157,319.438,417.785,179.628,16.415,151.562
C08066=1103.151,319.190,417.817,179.624,16.413,151.563
C08067=1103.145,318.943,417.849,179.620,16.411,151.563
C08068=1103.139,318.694,417.881,179.617,16.409,151.563
C08069=1103.134,318.447,417.913,179.614,16.407,151.563
C08070=1103.128,318.199,417.945,179.610,16.405,151.563
C08071=1103.123,317.951,417.976,179.607,16.403,151.564
C08072=1103.117,317.703,418.007,179.603,16.400,151.564
C08073=1103.111,317.455,418.039,179.600,16.398,151.564
C08074=1103.106,317.207,418.071,179.596,16.397,151.564
C08075=1103.098,316.824,418.120,179.591,16.394,151.565
C08076=1103.089,316.440,418.169,179.586,16.391,151.565
C08077=1103.080,316.058,418.218,179.581,16.387,151.565
C08078=1103.072,315.675,418.267,179.576,16.384,151.566
C08079=1103.066,315.426,418.298,179.572,16.382,151.566
C08080=1103.061,315.179,418.330,179.569,16.381,151.566
C08081=1103.054,314.931,418.361,179.566,16.379,151.566
C08082=1103.049,314.683,418.393,179.562,16.377,151.567
C08083=1103.043,314.434,418.424,179.559,16.376,151.567
C08084=1103.038,314.187,418.456,179.555,16.373,151.567
C08085=1103.031,313.940,418.487,179.552,16.372,151.568
C08086=1103.026,313.691,418.518,179.548,16.370,151.568
C08087=1103.020,313.443,418.550,179.545,16.368,151.568
C08088=1103.014,313.195,418.581,179.542,16.367,151.568
C08089=1103.009,312.947,418.612,179.538,16.365,151.569
C08090=1103.003,312.699,418.644,179.535,16.363,151.569
C08091=1102.997,312.451,418.675,179.531,16.361,151.569
C08092=1102.991,312.204,418.706,179.527,16.359,151.570
C08093=1102.985,311.955,418.737,179.525,16.358,151.570
C08094=1102.980,311.708,418.769,179.521,16.356,151.570
C08095=1102.974,311.459,418.800,179.517,16.354,151.571
C08096=1102.968,311.212,418.831,179.514,16.352,151.571
C08097=1102.963,310.963,418.862,179.510,16.350,151.571
C08098=1102.957,310.715,418.894,179.507,16.349,151.571
C08099=1102.951,310.467,418.924,179.504,16.348,151.572
C08100=1102.946,310.220,418.956,179.500,16.345,151.572
C08101=1102.939,309.971,418.987,179.497,16.344,151.572
C08102=1102.934,309.724,419.018,179.493,16.342,151.573
C08103=1102.928,309.476,419.049,179.490,16.340,151.573
C08104=1102.922,309.227,419.080,179.486,16.338,151.573
C08105=1102.917,308.980,419.112,179.483,16.337,151.573
C08106=1102.911,308.732,419.142,179.480,16.335,151.574
C08107=1102.906,308.484,419.174,179.476,16.334,151.574
C08108=1102.899,308.236,419.204,179.472,16.332,151.574
C08109=1102.894,307.988,419.235,179.469,16.330,151.575
C08110=1102.888,307.741,419.266,179.466,16.329,151.575
C08111=1102.882,307.492,419.298,179.462,16.327,151.575
C08112=1102.877,307.244,419.328,179.459,16.325,151.576
C08113=1102.871,306.996,419.359,179.455,16.323,151.576
C08114=1102.865,306.749,419.390,179.451,16.322,151.576
C08115=1102.860,306.500,419.421,179.448,16.319,151.577
C08116=1102.854,306.252,419.452,179.445,16.318,151.577
C08117=1102.849,306.004,419.483,179.441,16.317,151.577
C08118=1102.843,305.757,419.514,179.438,16.315,151.578
C08119=1102.838,305.508,419.545,179.434,16.313,151.578
C08120=1102.832,305.261,419.575,179.430,16.311,151.578
C08121=1102.826,305.012,419.606,179.428,16.310,151.579
C08122=1102.820,304.764,419.637,179.424,16.309,151.579
C08123=1102.814,304.516,419.667,179.420,16.307,151.579
C08124=1102.809,304.268,419.698,179.417,16.305,151.580
C08125=1102.803,304.021,419.729,179.413,16.303,151.580
C08126=1102.798,303.773,419.760,179.410,16.302,151.580
C08127=1102.789,303.392,419.807,179.405,16.299,151.581
C08128=1102.780,303.011,419.854,179.399,16.297,151.581
C08129=1102.772,302.631,419.901,179.394,16.294,151.582
C08130=1102.763,302.250,419.948,179.388,16.292,151.582
C08131=1102.758,302.001,419.978,179.385,16.290,151.583
C08132=1102.752,301.753,420.009,179.382,16.289,151.583
C08133=1102.747,301.505,420.039,179.378,16.287,151.583
C08134=1102.741,301.258,420.070,179.374,16.285,151.584
C08135=1102.736,301.009,420.101,179.371,16.284,151.584
C08136=1102.730,300.762,420.131,179.368,16.282,151.584
C08137=1102.724,300.514,420.161,179.364,16.281,151.585
C08138=1102.719,300.266,420.192,179.360,16.279,151.585
C08139=1102.713,300.018,420.223,179.358,16.278,151.585
C08140=1102.707,299.770,420.253,179.354,16.276,151.586
C08141=1102.702,299.522,420.284,179.350,16.274,151.586
C08142=1102.697,299.273,420.314,179.347,16.273,151.586
C08143=1102.691,299.026,420.344,179.344,16.272,151.587
C08144=1102.685,298.778,420.374,179.340,16.270,151.587
C08145=1102.680,298.530,420.405,179.336,16.268,151.588
C08146=1102.674,298.282,420.436,179.333,16.266,151.588
C08147=1102.669,298.033,420.465,179.330,16.265,151.588
C08148=1102.663,297.786,420.496,179.326,16.264,151.589
C08149=1102.657,297.538,420.526,179.322,16.262,151.589
C08150=1102.652,297.290,420.557,179.318,16.261,151.589
C08151=1102.646,297.040,420.587,179.316,16.260,151.590
C08152=1102.640,296.793,420.617,179.312,16.258,151.590
C08153=1102.634,296.545,420.648,179.308,16.257,151.591
C08154=1102.629,296.296,420.677,179.305,16.255,151.591
C08155=1102.623,296.049,420.708,179.301,16.254,151.591
C08156=1102.617,295.801,420.738,179.298,16.252,151.592
C08157=1102.612,295.552,420.768,179.294,16.251,151.592
C08158=1102.606,295.304,420.798,179.291,16.250,151.593
C08159=1102.600,295.056,420.828,179.287,16.248,151.593
C08160=1102.595,294.808,420.858,179.284,16.246,151.593
C08161=1102.589,294.560,420.888,179.280,16.245,151.594
C08162=1102.583,294.312,420.918,179.277,16.244,151.594
C08163=1102.577,294.064,420.948,179.273,16.242,151.594
C08164=1102.572,293.816,420.978,179.270,16.241,151.595
C08165=1102.566,293.568,421.008,179.266,16.240,151.595
C08166=1102.561,293.319,421.038,179.262,16.238,151.596
C08167=1102.555,293.072,421.068,179.258,16.237,151.596
C08168=1102.550,292.824,421.097,179.256,16.236,151.597
C08169=1102.544,292.576,421.128,179.252,16.234,151.597
C08170=1102.538,292.328,421.157,179.248,16.233,151.597
C08171=1102.533,292.080,421.188,179.245,16.231,151.598
C08172=1102.527,291.831,421.217,179.241,16.230,151.598
C08173=1102.522,291.583,421.247,179.237,16.228,151.599
C08174=1102.516,291.335,421.277,179.234,16.227,151.599
C08175=1102.510,291.087,421.307,179.231,16.226,151.599
C08176=1102.504,290.839,421.336,179.227,16.224,151.600
C08177=1102.498,290.591,421.366,179.224,16.223,151.600
C08178=1102.493,290.342,421.396,179.220,16.222,151.601
C08179=1102.485,289.976,421.440,179.215,16.220,151.601
C08180=1102.476,289.609,421.484,179.209,16.218,151.602
C08181=1102.468,289.243,421.528,179.205,16.216,151.602
C08182=1102.460,288.876,421.572,179.200,16.214,151.603
C08183=1102.454,288.628,421.602,179.196,16.213,151.604
C08184=1102.448,288.379,421.631,179.192,16.211,151.604
C08185=1102.442,288.131,421.660,179.189,16.211,151.605
C08186=1102.436,287.883,421.691,179.185,16.209,151.605
C08187=1102.431,287.635,421.720,179.181,16.208,151.605
C08188=1102.425,287.387,421.749,179.178,16.207,151.606
C08189=1102.419,287.138,421.779,179.174,16.205,151.606
C08190=1102.414,286.890,421.808,179.171,16.204,151.607
C08191=1102.409,286.642,421.838,179.167,16.203,151.607
C08192=1102.402,286.394,421.867,179.164,16.201,151.608
C08193=1102.397,286.146,421.897,179.160,16.201,151.608
C08194=1102.391,285.898,421.927,179.157,16.199,151.609
C08195=1102.385,285.649,421.956,179.153,16.198,151.609
C08196=1102.380,285.402,421.985,179.150,16.197,151.609
C08197=1102.374,285.153,422.015,179.146,16.195,151.610
C08198=1102.368,284.905,422.044,179.142,16.194,151.610
C08199=1102.363,284.657,422.073,179.139,16.193,151.611
C08200=1102.357,284.408,422.103,179.135,16.192,151.611
C08201=1102.352,284.161,422.132,179.132,16.191,151.612
C08202=1102.346,283.912,422.161,179.128,16.189,151.612
C08203=1102.341,283.664,422.191,179.124,16.188,151.613
C08204=1102.334,283.416,422.220,179.121,16.187,151.613
C08205=1102.329,283.168,422.249,179.117,16.186,151.613
C08206=1102.323,282.920,422.278,179.114,16.185,151.614
C08207=1102.318,282.671,422.308,179.111,16.183,151.614
C08208=1102.312,282.422,422.337,179.107,16.182,151.615
C08209=1102.307,282.175,422.366,179.104,16.181,151.615
C08210=1102.301,281.927,422.395,179.100,16.180,151.616
C08211=1102.296,281.678,422.425,179.097,16.179,151.616
C08212=1102.289,281.430,422.454,179.093,16.177,151.617
C08213=1102.285,281.182,422.483,179.089,16.176,151.617
C08214=1102.278,280.934,422.512,179.086,16.175,151.617
C08215=1102.273,280.685,422.541,179.082,16.174,151.618
C08216=1102.267,280.437,422.570,179.079,16.173,151.619
C08217=1102.261,280.189,422.599,179.075,16.172,151.619
C08218=1102.256,279.941,422.629,179.072,16.171,151.619
C08219=1102.250,279.692,422.657,179.068,16.169,151.620
C08220=1102.245,279.445,422.686,179.064,16.168,151.620
C08221=1102.239,279.196,422.715,179.061,16.167,151.621
C08222=1102.233,278.948,422.745,179.057,16.166,151.621
C08223=1102.227,278.699,422.773,179.054,16.165,151.622
C08224=1102.222,278.451,422.802,179.050,16.164,151.622
C08225=1102.216,278.203,422.831,179.047,16.163,151.623
C08226=1102.210,277.955,422.860,179.043,16.161,151.623
C08227=1102.205,277.707,422.889,179.039,16.160,151.624
C08228=1102.199,277.459,422.918,179.036,16.159,151.624
C08229=1102.194,277.210,422.947,179.032,16.158,151.625
C08230=1102.188,276.962,422.976,179.029,16.157,151.625
C08231=1102.179,276.605,423.017,179.024,16.156,151.626
C08232=1102.172,276.248,423.059,179.018,16.153,151.627
C08233=1102.163,275.890,423.100,179.013,16.152,151.627
C08234=1102.156,275.532,423.141,179.008,16.151,151.628
C08235=1102.149,275.284,423.170,179.005,16.150,151.629
C08236=1102.144,275.036,423.198,179.001,16.149,151.629
C08237=1102.138,274.788,423.228,178.997,16.148,151.630
C08238=1102.133,274.539,423.256,178.993,16.147,151.630
C08239=1102.127,274.291,423.285,178.990,16.146,151.631
C08240=1102.121,274.043,423.313,178.987,16.144,151.631
C08241=1102.116,273.795,423.342,178.983,16.143,151.632
C08242=1102.110,273.546,423.371,178.979,16.142,151.632
C08243=1102.104,273.299,423.399,178.975,16.141,151.633
C08244=1102.099,273.050,423.428,178.972,16.141,151.633
C08245=1102.093,272.801,423.456,178.968,16.139,151.634
C08246=1102.088,272.553,423.485,178.965,16.139,151.634
C08247=1102.082,272.305,423.514,178.961,16.137,151.635
C08248=1102.076,272.057,423.542,178.958,16.136,151.635
C08249=1102.070,271.808,423.571,178.954,16.135,151.636
C08250=1102.065,271.560,423.599,178.951,16.134,151.636
C08251=1102.059,271.312,423.627,178.947,16.133,151.637
C08252=1102.054,271.063,423.656,178.944,16.132,151.637
C08253=1102.048,270.815,423.685,178.940,16.131,151.638
C08254=1102.042,270.566,423.713,178.937,16.131,151.638
C08255=1102.037,270.318,423.741,178.933,16.129,151.639
C08256=1102.031,270.070,423.769,178.929,16.129,151.639
C08257=1102.025,269.822,423.798,178.925,16.127,151.640
C08258=1102.019,269.573,423.826,178.922,16.127,151.640
C08259=1102.014,269.325,423.854,178.918,16.125,151.641
C08260=1102.008,269.077,423.882,178.915,16.125,151.641
C08261=1102.003,268.829,423.910,178.911,16.124,151.642
C08262=1101.996,268.580,423.939,178.908,16.123,151.642
C08263=1101.991,268.332,423.967,178.904,16.122,151.643
C08264=1101.985,268.084,423.996,178.901,16.121,151.643
C08265=1101.980,267.836,424.024,178.897,16.120,151.644
C08266=1101.974,267.587,424.053,178.893,16.119,151.644
C08267=1101.969,267.339,424.081,178.889,16.118,151.645
C08268=1101.962,267.090,424.108,178.886,16.117,151.646
C08269=1101.957,266.842,424.136,178.882,16.116,151.646
C08270=1101.951,266.593,424.165,178.879,16.115,151.647
C08271=1101.946,266.345,424.192,178.875,16.114,151.647
C08272=1101.940,266.096,424.221,178.872,16.113,151.648
C08273=1101.935,265.848,424.249,178.868,16.112,151.648
C08274=1101.929,265.600,424.277,178.865,16.112,151.649
C08275=1101.923,265.352,424.305,178.861,16.110,151.649
C08276=1101.918,265.104,424.333,178.857,16.110,151.650
C08277=1101.912,264.855,424.361,178.853,16.108,151.650
C08278=1101.907,264.607,424.389,178.850,16.108,151.651
C08279=1101.901,264.358,424.418,178.846,16.107,151.651
C08280=1101.895,264.110,424.446,178.843,16.106,151.652
C08281=1101.889,263.861,424.474,178.840,16.105,151.652
C08282=1101.883,263.613,424.501,178.836,16.104,151.653
C08283=1101.876,263.258,424.541,178.830,16.103,151.654
C08284=1101.867,262.904,424.581,178.825,16.101,151.655
C08285=1101.859,262.549,424.621,178.820,16.100,151.655
C08286=1101.850,262.195,424.660,178.815,16.099,151.656
C08287=1101.845,261.946,424.688,178.811,16.099,151.657
C08288=1101.840,261.698,424.716,178.807,16.098,151.657
C08289=1101.833,261.450,424.743,178.804,16.097,151.658
C08290=1101.828,261.202,424.771,178.801,16.096,151.658
C08291=1101.822,260.952,424.799,178.797,16.095,151.659
C08292=1101.817,260.704,424.827,178.794,16.095,151.660
C08293=1101.811,260.457,424.854,178.790,16.094,151.660
C08294=1101.805,260.208,424.883,178.786,16.093,151.661
C08295=1101.800,259.959,424.910,178.782,16.092,151.661
C08296=1101.793,259.711,424.938,178.779,16.091,151.662
C08297=1101.788,259.463,424.966,178.776,16.091,151.662
C08298=1101.783,259.214,424.993,178.772,16.090,151.663
C08299=1101.776,258.965,425.021,178.768,16.089,151.664
C08300=1101.770,258.717,425.048,178.764,16.088,151.664
C08301=1101.765,258.469,425.075,178.761,16.087,151.665
C08302=1101.759,258.220,425.103,178.757,16.086,151.665
C08303=1101.754,257.972,425.131,178.754,16.086,151.666
C08304=1101.748,257.724,425.158,178.750,16.085,151.666
C08305=1101.742,257.475,425.186,178.746,16.084,151.667
C08306=1101.737,257.226,425.214,178.743,16.083,151.667
C08307=1101.731,256.978,425.240,178.739,16.082,151.668
C08308=1101.725,256.729,425.269,178.736,16.082,151.669
C08309=1101.719,256.481,425.295,178.732,16.081,151.669
C08310=1101.714,256.233,425.323,178.729,16.080,151.670
C08311=1101.708,255.985,425.350,178.725,16.080,151.670
C08312=1101.702,255.736,425.378,178.721,16.078,151.671
C08313=1101.697,255.487,425.405,178.718,16.078,151.671
C08314=1101.691,255.239,425.433,178.714,16.077,151.672
C08315=1101.686,254.991,425.460,178.711,16.076,151.673
C08316=1101.679,254.742,425.488,178.707,16.076,151.673
C08317=1101.674,254.494,425.515,178.703,16.075,151.674
C08318=1101.668,254.245,425.542,178.700,16.074,151.674
C08319=1101.663,253.997,425.570,178.696,16.073,151.675
C08320=1101.657,253.748,425.597,178.693,16.072,151.675
C08321=1101.652,253.500,425.624,178.688,16.071,151.676
C08322=1101.646,253.252,425.651,178.685,16.071,151.677
C08323=1101.641,253.003,425.678,178.682,16.070,151.677
C08324=1101.635,252.755,425.705,178.678,16.069,151.678
C08325=1101.629,252.506,425.733,178.674,16.069,151.678
C08326=1101.623,252.258,425.760,178.670,16.067,151.679
C08327=1101.618,252.009,425.787,178.667,16.067,151.679
C08328=1101.612,251.761,425.814,178.664,16.066,151.680
C08329=1101.607,251.513,425.842,178.660,16.065,151.681
C08330=1101.601,251.264,425.869,178.656,16.065,151.681
C08331=1101.596,251.015,425.896,178.653,16.064,151.682
C08332=1101.590,250.766,425.923,178.649,16.063,151.682
C08333=1101.585,250.518,425.950,178.646,16.062,151.683
C08334=1101.579,250.269,425.977,178.642,16.061,151.683
C08335=1101.571,249.913,426.016,178.637,16.060,151.684
C08336=1101.563,249.555,426.055,178.632,16.060,151.685
C08337=1101.555,249.198,426.094,178.627,16.058,151.686
C08338=1101.547,248.840,426.132,178.622,16.057,151.687
C08339=1101.541,248.592,426.160,178.618,16.057,151.687
C08340=1101.536,248.343,426.187,178.614,16.055,151.688
C08341=1101.530,248.095,426.213,178.611,16.055,151.689
C08342=1101.525,247.846,426.241,178.607,16.054,151.689
C08343=1101.519,247.598,426.267,178.604,16.053,151.690
C08344=1101.514,247.349,426.295,178.600,16.053,151.690
C08345=1101.508,247.101,426.321,178.596,16.052,151.691
C08346=1101.502,246.852,426.348,178.593,16.051,151.691
C08347=1101.497,246.604,426.375,178.590,16.051,151.692
C08348=1101.492,246.355,426.402,178.585,16.050,151.693
C08349=1101.486,246.107,426.428,178.582,16.049,151.693
C08350=1101.479,245.858,426.455,178.579,16.049,151.694
C08351=1101.474,245.609,426.481,178.575,16.048,151.694
C08352=1101.468,245.361,426.508,178.571,16.047,151.695
C08353=1101.463,245.112,426.535,178.567,16.046,151.695
C08354=1101.457,244.864,426.562,178.564,16.046,151.696
C08355=1101.452,244.615,426.589,178.561,16.045,151.697
C08356=1101.446,244.367,426.615,178.557,16.044,151.697
C08357=1101.440,244.119,426.642,178.553,16.044,151.698
C08358=1101.435,243.870,426.669,178.550,16.043,151.698
C08359=1101.430,243.621,426.695,178.546,16.042,151.699
C08360=1101.424,243.373,426.722,178.542,16.042,151.700
C08361=1101.418,243.124,426.748,178.539,16.041,151.700
C08362=1101.412,242.876,426.775,178.535,16.041,151.701
C08363=1101.407,242.627,426.801,178.532,16.040,151.702
C08364=1101.401,242.379,426.828,178.528,16.039,151.702
C08365=1101.395,242.130,426.854,178.524,16.039,151.703
C08366=1101.389,241.882,426.881,178.521,16.038,151.703
C08367=1101.384,241.633,426.907,178.517,16.038,151.704
C08368=1101.378,241.384,426.933,178.513,16.037,151.705
C08369=1101.372,241.136,426.960,178.510,16.036,151.705
C08370=1101.367,240.887,426.987,178.507,16.036,151.706
C08371=1101.362,240.638,427.013,178.503,16.035,151.706
C08372=1101.356,240.390,427.040,178.499,16.034,151.707
C08373=1101.350,240.142,427.067,178.496,16.034,151.708
C08374=1101.345,239.893,427.092,178.492,16.034,151.708
C08375=1101.338,239.645,427.119,178.488,16.032,151.709
C08376=1101.333,239.396,427.144,178.485,16.032,151.709
C08377=1101.327,239.147,427.171,178.482,16.032,151.710
C08378=1101.321,238.899,427.198,178.478,16.031,151.711
C08379=1101.316,238.650,427.224,178.474,16.030,151.711
C08380=1101.310,238.402,427.250,178.471,16.030,151.712
C08381=1101.305,238.153,427.276,178.467,16.029,151.713
C08382=1101.299,237.904,427.303,178.463,16.028,151.713
C08383=1101.294,237.656,427.328,178.460,16.028,151.714
C08384=1101.288,237.408,427.355,178.457,16.028,151.714
C08385=1101.283,237.159,427.381,178.453,16.026,151.715
C08386=1101.277,236.910,427.408,178.449,16.026,151.716
C08387=1101.268,236.546,427.445,178.444,16.025,151.716
C08388=1101.260,236.182,427.484,178.438,16.024,151.717
C08389=1101.252,235.817,427.523,178.433,16.023,151.718
C08390=1101.244,235.453,427.560,178.428,16.023,151.719
C08391=1101.238,235.205,427.587,178.424,16.022,151.720
C08392=1101.232,234.956,427.613,178.421,16.022,151.720
C08393=1101.227,234.707,427.639,178.418,16.021,151.721
C08394=1101.222,234.459,427.665,178.413,16.020,151.722
C08395=1101.216,234.210,427.691,178.410,16.020,151.722
C08396=1101.210,233.962,427.716,178.406,16.020,151.723
C08397=1101.204,233.713,427.743,178.403,16.019,151.723
C08398=1101.199,233.464,427.769,178.399,16.018,151.724
C08399=1101.193,233.215,427.795,178.396,16.018,151.725
C08400=1101.187,232.968,427.820,178.392,16.017,151.725
C08401=1101.182,232.719,427.846,178.389,16.017,151.726
C08402=1101.176,232.470,427.872,178.385,16.016,151.727
C08403=1101.171,232.221,427.898,178.381,16.015,151.727
C08404=1101.164,231.973,427.924,178.378,16.015,151.728
C08405=1101.160,231.725,427.950,178.375,16.015,151.728
C08406=1101.154,231.476,427.976,178.371,16.014,151.729
C08407=1101.149,231.227,428.002,178.367,16.013,151.730
C08408=1101.142,230.978,428.027,178.364,16.013,151.730
C08409=1101.137,230.729,428.053,178.360,16.012,151.731
C08410=1101.132,230.481,428.079,178.356,16.011,151.732
C08411=1101.126,230.233,428.105,178.353,16.011,151.732
C08412=1101.120,229.984,428.130,178.350,16.011,151.733
C08413=1101.114,229.735,428.156,178.345,16.010,151.733
C08414=1101.108,229.486,428.182,178.342,16.010,151.734
C08415=1101.104,229.238,428.207,178.339,16.009,151.735
C08416=1101.097,228.989,428.233,178.335,16.009,151.735
C08417=1101.092,228.740,428.259,178.332,16.009,151.736
C08418=1101.086,228.492,428.284,178.327,16.008,151.737
C08419=1101.081,228.243,428.309,178.324,16.007,151.737
C08420=1101.075,227.995,428.335,178.321,16.007,151.738
C08421=1101.069,227.746,428.361,178.317,16.006,151.738
C08422=1101.063,227.497,428.386,178.313,16.006,151.739
C08423=1101.058,227.249,428.412,178.310,16.006,151.740
C08424=1101.052,227.000,428.437,178.306,16.005,151.740
C08425=1101.046,226.751,428.463,178.303,16.005,151.741
C08426=1101.040,226.502,428.488,178.299,16.004,151.742
C08427=1101.035,226.254,428.514,178.295,16.003,151.742
C08428=1101.029,226.005,428.539,178.292,16.003,151.743
C08429=1101.024,225.756,428.565,178.289,16.003,151.744
C08430=1101.018,225.508,428.590,178.285,16.002,151.744
C08431=1101.013,225.259,428.616,178.281,16.001,151.745
C08432=1101.006,225.011,428.641,178.278,16.001,151.745
C08433=1101.002,224.762,428.667,178.274,16.001,151.746
C08434=1100.995,224.514,428.692,178.271,16.000,151.747
C08435=1100.990,224.264,428.717,178.267,15.999,151.747
C08436=1100.985,224.016,428.742,178.263,15.999,151.748
C08437=1100.979,223.767,428.768,178.260,15.999,151.749
C08438=1100.973,223.519,428.794,178.256,15.999,151.749
C08439=1100.965,223.146,428.832,178.251,15.998,151.750
C08440=1100.957,222.773,428.869,178.246,15.997,151.751
C08441=1100.948,222.401,428.907,178.240,15.996,151.752
C08442=1100.940,222.028,428.945,178.235,15.996,151.753
C08443=1100.934,221.780,428.970,178.231,15.995,151.754
C08444=1100.928,221.530,428.995,178.228,15.995,151.754
C08445=1100.923,221.282,429.020,178.224,15.994,151.755
C08446=1100.917,221.033,429.046,178.221,15.994,151.756
C08447=1100.911,220.785,429.071,178.217,15.994,151.756
C08448=1100.906,220.536,429.096,178.213,15.993,151.757
C08449=1100.900,220.287,429.121,178.210,15.992,151.758
C08450=1100.894,220.038,429.145,178.206,15.992,151.758
C08451=1100.888,219.790,429.171,178.203,15.992,151.759
C08452=1100.883,219.541,429.196,178.200,15.992,151.760
C08453=1100.877,219.292,429.221,178.196,15.990,151.760
C08454=1100.871,219.044,429.246,178.192,15.990,151.761
C08455=1100.866,218.795,429.271,178.189,15.990,151.762
C08456=1100.860,218.546,429.296,178.185,15.990,151.762
C08457=1100.855,218.298,429.321,178.182,15.989,151.763
C08458=1100.849,218.049,429.346,178.179,15.989,151.763
C08459=1100.843,217.801,429.371,178.174,15.988,151.764
C08460=1100.837,217.551,429.396,178.171,15.988,151.765
C08461=1100.833,217.303,429.421,178.167,15.987,151.765
C08462=1100.827,217.054,429.446,178.164,15.987,151.766
C08463=1100.821,216.806,429.471,178.161,15.987,151.767
C08464=1100.815,216.557,429.495,178.157,15.987,151.767
C08465=1100.810,216.308,429.520,178.153,15.986,151.768
C08466=1100.804,216.059,429.545,178.150,15.985,151.769
C08467=1100.799,215.810,429.570,178.146,15.985,151.769
C08468=1100.793,215.562,429.595,178.143,15.985,151.770
C08469=1100.788,215.313,429.619,178.139,15.985,151.771
C08470=1100.781,215.065,429.645,178.136,15.984,151.771
C08471=1100.776,214.816,429.669,178.132,15.983,151.772
C08472=1100.770,214.567,429.694,178.128,15.983,151.773
C08473=1100.765,214.319,429.719,178.125,15.983,151.773
C08474=1100.759,214.069,429.743,178.121,15.982,151.774
C08475=1100.754,213.821,429.768,178.118,15.982,151.774
C08476=1100.748,213.572,429.793,178.115,15.982,151.775
C08477=1100.743,213.323,429.818,178.110,15.981,151.776
C08478=1100.737,213.074,429.842,178.107,15.980,151.776
C08479=1100.731,212.825,429.867,178.104,15.980,151.777
C08480=1100.726,212.577,429.892,178.100,15.980,151.778
C08481=1100.720,212.328,429.916,178.097,15.980,151.778
C08482=1100.715,212.080,429.940,178.093,15.980,151.779
C08483=1100.709,211.830,429.965,178.090,15.979,151.780
C08484=1100.703,211.582,429.990,178.086,15.978,151.780
C08485=1100.698,211.334,430.014,178.082,15.978,151.781
C08486=1100.692,211.084,430.039,178.079,15.978,151.782
C08487=1100.687,210.836,430.063,178.075,15.978,151.782
C08488=1100.680,210.587,430.087,178.072,15.977,151.783
C08489=1100.674,210.339,430.112,178.069,15.977,151.784
C08490=1100.668,210.090,430.137,178.065,15.977,151.784
C08491=1100.661,209.721,430.173,178.060,15.976,151.785
C08492=1100.652,209.352,430.209,178.054,15.975,151.786
C08493=1100.644,208.983,430.246,178.049,15.975,151.787
C08494=1100.636,208.614,430.282,178.044,15.974,151.788
C08495=1100.613,207.607,430.379,178.006,15.964,151.794
C08496=1100.607,207.359,430.403,178.002,15.965,151.795
C08497=1100.602,207.110,430.427,177.998,15.965,151.796
C08498=1100.596,206.861,430.452,177.995,15.965,151.796
C08499=1100.590,206.613,430.476,177.991,15.966,151.797
C08500=1100.584,206.364,430.500,177.987,15.966,151.798
C08501=1100.579,206.116,430.524,177.984,15.967,151.799
C08502=1100.572,205.867,430.548,177.980,15.968,151.800
C08503=1100.567,205.618,430.572,177.976,15.968,151.801
C08504=1100.562,205.369,430.596,177.972,15.968,151.802
C08505=1100.556,205.120,430.621,177.968,15.969,151.803
C08506=1100.550,204.871,430.644,177.964,15.969,151.804
C08507=1100.545,204.623,430.668,177.961,15.970,151.805
C08508=1100.540,204.374,430.693,177.957,15.970,151.805
C08509=1100.534,204.125,430.716,177.954,15.971,151.806
C08510=1100.528,203.876,430.740,177.950,15.971,151.807
C08511=1100.522,203.628,430.764,177.946,15.972,151.808
C08512=1100.517,203.379,430.788,177.942,15.972,151.809
C08513=1100.512,203.130,430.812,177.939,15.973,151.810
C08514=1100.505,202.881,430.836,177.935,15.973,151.811
C08515=1100.500,202.632,430.860,177.931,15.974,151.812
C08516=1100.494,202.384,430.884,177.927,15.974,151.812
C08517=1100.489,202.135,430.907,177.924,15.974,151.813
C08518=1100.482,201.886,430.931,177.920,15.975,151.814
C08519=1100.477,201.637,430.955,177.916,15.976,151.815
C08520=1100.471,201.388,430.978,177.912,15.976,151.816
C08521=1100.466,201.140,431.003,177.909,15.977,151.817
C08522=1100.459,200.891,431.027,177.905,15.977,151.818
C08523=1100.454,200.642,431.050,177.902,15.978,151.819
C08524=1100.448,200.393,431.074,177.898,15.978,151.820
C08525=1100.442,200.144,431.097,177.894,15.979,151.820
C08526=1100.437,199.896,431.121,177.890,15.979,151.821
C08527=1100.430,199.647,431.145,177.886,15.979,151.822
C08528=1100.425,199.398,431.169,177.882,15.980,151.823
C08529=1100.419,199.149,431.192,177.879,15.981,151.824
C08530=1100.414,198.900,431.216,177.875,15.981,151.825
C08531=1100.408,198.652,431.240,177.872,15.982,151.826
C08532=1100.402,198.402,431.263,177.868,15.982,151.827
C08533=1100.397,198.154,431.287,177.864,15.982,151.827
C08534=1100.391,197.905,431.310,177.861,15.983,151.828
C08535=1100.385,197.657,431.334,177.857,15.984,151.829
C08536=1100.380,197.407,431.357,177.853,15.984,151.830
C08537=1100.374,197.159,431.381,177.849,15.984,151.831
C08538=1100.369,196.910,431.404,177.845,15.985,151.832
C08539=1100.362,196.661,431.428,177.842,15.986,151.833
C08540=1100.357,196.412,431.451,177.839,15.986,151.834
C08541=1100.351,196.163,431.476,177.835,15.986,151.834
C08542=1100.346,195.914,431.499,177.831,15.986,151.835
C08543=1100.340,195.666,431.522,177.827,15.987,151.836
C08544=1100.334,195.417,431.546,177.824,15.988,151.837
C08545=1100.329,195.168,431.569,177.820,15.988,151.838
C08546=1100.323,194.919,431.592,177.817,15.988,151.839
C08547=1100.318,194.671,431.616,177.813,15.989,151.840
C08548=1100.312,194.422,431.639,177.809,15.989,151.840
C08549=1100.306,194.172,431.662,177.806,15.990,151.841
C08550=1100.300,193.924,431.686,177.802,15.990,151.842
C08551=1100.295,193.675,431.709,177.798,15.990,151.843
C08552=1100.289,193.426,431.732,177.794,15.991,151.844
C08553=1100.283,193.177,431.756,177.791,15.992,151.845
C08554=1100.278,192.928,431.780,177.788,15.992,151.846
C08555=1100.272,192.679,431.803,177.784,15.993,151.846
C08556=1100.266,192.407,431.828,177.780,15.993,151.847
C08557=1100.260,192.133,431.854,177.776,15.993,151.848
C08558=1100.253,191.861,431.879,177.772,15.994,151.849
C08559=1100.248,191.588,431.904,177.768,15.995,151.850
C08560=1100.242,191.339,431.928,177.764,15.994,151.851
C08561=1100.237,191.090,431.951,177.761,15.995,151.852
C08562=1100.231,190.841,431.974,177.757,15.995,151.853
C08563=1100.225,190.592,431.997,177.754,15.996,151.853
C08564=1100.219,190.343,432.020,177.750,15.996,151.854
C08565=1100.214,190.094,432.044,177.746,15.997,151.855
C08566=1100.209,189.845,432.067,177.742,15.997,151.856
C08567=1100.203,189.597,432.090,177.739,15.997,151.857
C08568=1100.197,189.348,432.113,177.736,15.998,151.858
C08569=1100.191,189.099,432.136,177.732,15.998,151.858
C08570=1100.186,188.850,432.160,177.728,15.999,151.859
C08571=1100.180,188.601,432.183,177.725,15.999,151.860
C08572=1100.175,188.352,432.206,177.721,16.000,151.861
C08573=1100.169,188.103,432.228,177.718,15.999,151.862
C08574=1100.163,187.854,432.251,177.714,16.000,151.862
C08575=1100.158,187.605,432.275,177.710,16.000,151.863
C08576=1100.153,187.357,432.298,177.707,16.000,151.864
C08577=1100.147,187.108,432.320,177.704,16.001,151.865
C08578=1100.142,186.859,432.343,177.700,16.002,151.866
C08579=1100.136,186.610,432.366,177.696,16.002,151.867
C08580=1100.130,186.361,432.389,177.692,16.002,151.867
C08581=1100.125,186.112,432.412,177.689,16.002,151.868
C08582=1100.120,185.863,432.436,177.686,16.003,151.869
C08583=1100.114,185.614,432.459,177.682,16.003,151.870
C08584=1100.109,185.366,432.481,177.678,16.003,151.871
C08585=1100.103,185.117,432.504,177.674,16.004,151.872
C08586=1100.098,184.868,432.527,177.671,16.005,151.872
C08587=1100.092,184.619,432.549,177.668,16.005,151.873
C08588=1100.085,184.370,432.572,177.664,16.005,151.874
C08589=1100.080,184.121,432.595,177.660,16.005,151.875
C08590=1100.074,183.873,432.618,177.657,16.006,151.876
C08591=1100.068,183.624,432.641,177.654,16.006,151.876
C08592=1100.062,183.375,432.664,177.650,16.007,151.877
C08593=1100.057,183.125,432.686,177.646,16.007,151.878
C08594=1100.050,182.877,432.708,177.643,16.008,151.879
C08595=1100.045,182.628,432.731,177.639,16.008,151.880
C08596=1100.039,182.379,432.754,177.635,16.008,151.881
C08597=1100.033,182.130,432.777,177.632,16.008,151.881
C08598=1100.028,181.880,432.799,177.629,16.009,151.882
C08599=1100.022,181.633,432.821,177.625,16.010,151.883
C08600=1100.016,181.384,432.844,177.621,16.010,151.884
C08601=1100.011,181.135,432.867,177.617,16.010,151.885
C08602=1100.005,180.885,432.889,177.614,16.011,151.886
C08603=1099.999,180.636,432.912,177.611,16.011,151.886
C08604=1099.993,180.388,432.935,177.607,16.011,151.887
C08605=1099.987,180.139,432.958,177.603,16.011,151.888
C08606=1099.982,179.889,432.980,177.600,16.012,151.889
C08607=1099.977,179.641,433.002,177.596,16.013,151.890
C08608=1099.970,179.393,433.025,177.593,16.013,151.890
C08609=1099.965,179.143,433.047,177.589,16.013,151.891
C08610=1099.959,178.894,433.070,177.586,16.014,151.892
C08611=1099.953,178.645,433.093,177.582,16.014,151.893
C08612=1099.947,178.396,433.115,177.579,16.014,151.894
C08613=1099.942,178.148,433.137,177.576,16.015,151.895
C08614=1099.937,177.898,433.159,177.572,16.015,151.895
C08615=1099.931,177.649,433.182,177.568,16.016,151.896
C08616=1099.924,177.401,433.205,177.565,16.015,151.897
C08617=1099.919,177.151,433.227,177.562,16.017,151.898
C08618=1099.914,176.903,433.249,177.558,16.016,151.898
C08619=1099.908,176.654,433.271,177.554,16.017,151.899
C08620=1099.902,176.381,433.296,177.551,16.017,151.900
C08621=1099.895,176.107,433.321,177.547,16.018,151.901
C08622=1099.889,175.834,433.345,177.543,16.018,151.902
C08623=1099.883,175.560,433.370,177.539,16.018,151.903
C08624=1099.877,175.311,433.391,177.535,16.018,151.904
C08625=1099.871,175.062,433.414,177.533,16.019,151.904
C08626=1099.866,174.813,433.437,177.529,16.019,151.905
C08627=1099.860,174.565,433.459,177.525,16.019,151.906
C08628=1099.855,174.315,433.481,177.522,16.019,151.907
C08629=1099.849,174.066,433.502,177.519,16.020,151.908
C08630=1099.843,173.817,433.525,177.515,16.020,151.908
C08631=1099.838,173.569,433.547,177.511,16.021,151.909
C08632=1099.832,173.320,433.570,177.508,16.021,151.910
C08633=1099.826,173.070,433.592,177.505,16.021,151.911
C08634=1099.821,172.822,433.614,177.501,16.022,151.911
C08635=1099.815,172.573,433.636,177.497,16.022,151.912
C08636=1099.809,172.324,433.658,177.495,16.022,151.913
C08637=1099.804,172.075,433.680,177.491,16.023,151.914
C08638=1099.798,171.826,433.702,177.487,16.023,151.915
C08639=1099.793,171.577,433.725,177.484,16.023,151.915
C08640=1099.787,171.328,433.746,177.481,16.023,151.916
C08641=1099.781,171.079,433.769,177.477,16.024,151.917
C08642=1099.775,170.830,433.791,177.474,16.024,151.918
C08643=1099.770,170.581,433.812,177.470,16.024,151.918
C08644=1099.764,170.332,433.834,177.467,16.024,151.919
C08645=1099.759,170.084,433.857,177.463,16.025,151.920
C08646=1099.754,169.834,433.879,177.460,16.025,151.921
C08647=1099.748,169.585,433.901,177.457,16.025,151.921
C08648=1099.743,169.336,433.922,177.453,16.025,151.922
C08649=1099.737,169.087,433.944,177.450,16.026,151.923
C08650=1099.731,168.839,433.967,177.446,16.026,151.924
C08651=1099.725,168.590,433.988,177.443,16.026,151.924
C08652=1099.720,168.340,434.010,177.440,16.026,151.925
C08653=1099.714,168.092,434.032,177.436,16.026,151.926
C08654=1099.709,167.842,434.054,177.433,16.027,151.927
C08655=1099.703,167.594,434.075,177.430,16.027,151.927
C08656=1099.698,167.345,434.098,177.426,16.027,151.928
C08657=1099.692,167.096,434.119,177.422,16.027,151.929
C08658=1099.687,166.847,434.142,177.420,16.028,151.930
C08659=1099.680,166.597,434.163,177.416,16.028,151.930
C08660=1099.676,166.349,434.185,177.413,16.028,151.931
C08661=1099.669,166.099,434.207,177.409,16.028,151.932
C08662=1099.665,165.851,434.229,177.406,16.028,151.933
C08663=1099.658,165.601,434.250,177.402,16.029,151.933
C08664=1099.654,165.353,434.272,177.399,16.029,151.934
C08665=1099.647,165.103,434.294,177.396,16.029,151.935
C08666=1099.643,164.855,434.316,177.392,16.029,151.936
C08667=1099.636,164.605,434.337,177.389,16.029,151.936
C08668=1099.632,164.357,434.359,177.385,16.029,151.937
C08669=1099.625,164.107,434.381,177.383,16.030,151.938
C08670=1099.621,163.859,434.403,177.379,16.030,151.938
C08671=1099.614,163.609,434.424,177.375,16.030,151.939
C08672=1099.609,163.361,434.446,177.373,16.030,151.940
C08673=1099.604,163.112,434.467,177.369,16.030,151.941
C08674=1099.598,162.863,434.489,177.366,16.030,151.941
C08675=1099.593,162.614,434.511,177.362,16.030,151.942
C08676=1099.587,162.364,434.532,177.359,16.031,151.943
C08677=1099.582,162.116,434.553,177.356,16.031,151.944
C08678=1099.576,161.866,434.575,177.352,16.031,151.944
C08679=1099.571,161.618,434.597,177.349,16.031,151.945
C08680=1099.565,161.368,434.618,177.346,16.031,151.946
C08681=1099.560,161.120,434.640,177.342,16.031,151.946
C08682=1099.554,160.870,434.662,177.339,16.032,151.947
C08683=1099.548,160.622,434.683,177.336,16.032,151.948
C08684=1099.542,160.348,434.707,177.332,16.032,151.949
C08685=1099.536,160.073,434.730,177.329,16.032,151.950
C08686=1099.530,159.800,434.753,177.325,16.032,151.950
C08687=1099.523,159.526,434.776,177.321,16.033,151.951
C08688=1099.518,159.278,434.798,177.318,16.033,151.952
C08689=1099.512,159.028,434.820,177.315,16.033,151.953
C08690=1099.506,158.780,434.841,177.311,16.033,151.953
C08691=1099.501,158.530,434.862,177.308,16.033,151.954
C08692=1099.495,158.281,434.883,177.305,16.033,151.955
C08693=1099.489,158.032,434.905,177.302,16.033,151.955
C08694=1099.483,157.784,434.926,177.298,16.033,151.956
C08695=1099.479,157.534,434.947,177.295,16.034,151.957
C08696=1099.473,157.285,434.969,177.292,16.034,151.958
C08697=1099.467,157.037,434.990,177.288,16.034,151.958
C08698=1099.461,156.787,435.011,177.285,16.034,151.959
C08699=1099.456,156.538,435.032,177.282,16.035,151.960
C08700=1099.449,156.289,435.054,177.278,16.035,151.960
C08701=1099.444,156.040,435.075,177.275,16.035,151.961
C08702=1099.439,155.791,435.096,177.272,16.035,151.962
C08703=1099.433,155.542,435.118,177.269,16.035,151.962
C08704=1099.427,155.293,435.138,177.265,16.035,151.963
C08705=1099.422,155.045,435.159,177.262,16.035,151.964
C08706=1099.417,154.794,435.181,177.259,16.035,151.965
C08707=1099.411,154.546,435.202,177.255,16.035,151.965
C08708=1099.405,154.297,435.224,177.252,16.036,151.966
C08709=1099.400,154.048,435.244,177.249,16.036,151.967
C08710=1099.394,153.799,435.266,177.245,16.036,151.968
C08711=1099.388,153.549,435.287,177.243,16.036,151.968
C08712=1099.383,153.301,435.308,177.239,16.036,151.969
C08713=1099.377,153.052,435.328,177.236,16.036,151.970
C08714=1099.371,152.802,435.350,177.233,16.037,151.970
C08715=1099.365,152.554,435.370,177.229,16.037,151.971
C08716=1099.360,152.305,435.391,177.226,16.036,151.972
C08717=1099.354,152.055,435.412,177.223,16.037,151.972
C08718=1099.348,151.807,435.433,177.220,16.037,151.973
C08719=1099.343,151.558,435.454,177.216,16.037,151.974
C08720=1099.337,151.308,435.475,177.214,16.038,151.974
C08721=1099.332,151.059,435.496,177.210,16.037,151.975
C08722=1099.326,150.810,435.517,177.207,16.037,151.976
C08723=1099.320,150.561,435.538,177.204,16.038,151.976
C08724=1099.315,150.312,435.559,177.200,16.038,151.977
C08725=1099.309,150.063,435.580,177.197,16.037,151.978
C08726=1099.303,149.814,435.601,177.194,16.038,151.978
C08727=1099.298,149.564,435.622,177.191,16.038,151.979
C08728=1099.293,149.316,435.643,177.187,16.037,151.980
C08729=1099.287,149.067,435.663,177.185,16.038,151.981
C08730=1099.281,148.817,435.684,177.181,16.038,151.981
C08731=1099.275,148.569,435.705,177.178,16.038,151.982
C08732=1099.270,148.320,435.726,177.175,16.038,151.983
C08733=1099.264,148.070,435.747,177.172,16.038,151.983
C08734=1099.259,147.821,435.768,177.168,16.038,151.984
C08735=1099.253,147.573,435.788,177.166,16.038,151.985
C08736=1099.247,147.323,435.808,177.162,16.038,151.985
C08737=1099.241,147.074,435.829,177.158,16.038,151.986
C08738=1099.236,146.825,435.851,177.156,16.039,151.987
C08739=1099.230,146.576,435.870,177.152,16.039,151.987
C08740=1099.225,146.327,435.891,177.149,16.039,151.988
C08741=1099.219,146.077,435.912,177.146,16.039,151.989
C08742=1099.213,145.829,435.933,177.143,16.039,151.989
C08743=1099.207,145.580,435.953,177.139,16.039,151.990
C08744=1099.202,145.331,435.974,177.137,16.039,151.991
C08745=1099.196,145.081,435.995,177.133,16.039,151.991
C08746=1099.191,144.832,436.015,177.130,16.038,151.992
C08747=1099.185,144.583,436.035,177.127,16.039,151.993
C08748=1099.179,144.310,436.059,177.124,16.039,151.993
C08749=1099.172,144.036,436.081,177.120,16.039,151.994
C08750=1099.166,143.762,436.103,177.116,16.039,151.995
C08751=1099.160,143.487,436.126,177.113,16.039,151.996
C08752=1099.154,143.239,436.146,177.110,16.039,151.996
C08753=1099.149,142.989,436.167,177.107,16.039,151.997
C08754=1099.143,142.740,436.188,177.104,16.039,151.997
C08755=1099.138,142.490,436.208,177.101,16.040,151.998
C08756=1099.132,142.242,436.228,177.098,16.039,151.999
C08757=1099.127,141.992,436.249,177.094,16.039,152.000
C08758=1099.121,141.743,436.269,177.092,16.039,152.000
C08759=1099.115,141.494,436.290,177.088,16.039,152.001
C08760=1099.109,141.245,436.311,177.085,16.039,152.001
C08761=1099.104,140.996,436.331,177.082,16.039,152.002
C08762=1099.098,140.747,436.351,177.079,16.039,152.003
C08763=1099.093,140.498,436.372,177.075,16.039,152.003
C08764=1099.087,140.249,436.391,177.073,16.039,152.004
C08765=1099.082,140.000,436.412,177.069,16.039,152.005
C08766=1099.075,139.750,436.432,177.066,16.039,152.005
C08767=1099.070,139.501,436.453,177.063,16.039,152.006
C08768=1099.065,139.252,436.473,177.060,16.039,152.007
C08769=1099.059,139.003,436.493,177.057,16.039,152.007
C08770=1099.054,138.754,436.514,177.054,16.039,152.008
C08771=1099.048,138.505,436.534,177.050,16.039,152.008
C08772=1099.042,138.256,436.554,177.048,16.039,152.009
C08773=1099.036,138.007,436.574,177.044,16.039,152.010
C08774=1099.031,137.758,436.595,177.041,16.038,152.010
C08775=1099.024,137.509,436.615,177.038,16.039,152.011
C08776=1099.019,137.259,436.635,177.035,16.039,152.012
C08777=1099.013,137.010,436.655,177.032,16.039,152.012
C08778=1099.008,136.761,436.675,177.029,16.039,152.013
C08779=1099.002,136.512,436.695,177.026,16.038,152.013
C08780=1098.996,136.263,436.715,177.023,16.039,152.014
C08781=1098.991,136.014,436.736,177.020,16.039,152.015
C08782=1098.985,135.765,436.755,177.017,16.038,152.015
C08783=1098.980,135.516,436.776,177.014,16.039,152.016
C08784=1098.974,135.267,436.796,177.010,16.038,152.017
C08785=1098.969,135.018,436.816,177.007,16.038,152.017
C08786=1098.963,134.769,436.836,177.004,16.039,152.018
C08787=1098.958,134.519,436.856,177.001,16.038,152.019
C08788=1098.951,134.270,436.876,176.999,16.038,152.019
C08789=1098.945,134.021,436.896,176.995,16.038,152.020
C08790=1098.940,133.771,436.916,176.992,16.038,152.020
C08791=1098.934,133.522,436.936,176.989,16.038,152.021
C08792=1098.929,133.273,436.957,176.986,16.038,152.022
C08793=1098.923,133.024,436.976,176.983,16.038,152.022
C08794=1098.917,132.775,436.996,176.980,16.038,152.023
C08795=1098.912,132.526,437.016,176.977,16.037,152.023
C08796=1098.906,132.277,437.036,176.974,16.038,152.024
C08797=1098.900,132.028,437.055,176.971,16.038,152.025
C08798=1098.895,131.778,437.076,176.968,16.037,152.025
C08799=1098.890,131.529,437.095,176.965,16.037,152.026
C08800=1098.884,131.280,437.115,176.962,16.037,152.026
C08801=1098.878,131.031,437.135,176.959,16.038,152.027
C08802=1098.873,130.782,437.155,176.956,16.037,152.028
C08803=1098.867,130.533,437.175,176.952,16.037,152.028
C08804=1098.861,130.283,437.194,176.950,16.037,152.029
C08805=1098.855,130.035,437.214,176.946,16.037,152.030
C08806=1098.849,129.786,437.234,176.944,16.037,152.030
C08807=1098.844,129.536,437.254,176.941,16.037,152.031
C08808=1098.838,129.287,437.274,176.937,16.036,152.031
C08809=1098.832,129.038,437.293,176.935,16.037,152.032
C08810=1098.826,128.789,437.313,176.931,16.037,152.033
C08811=1098.821,128.540,437.332,176.928,16.036,152.033
C08812=1098.816,128.325,437.350,176.926,16.036,152.034
C08813=1098.811,128.110,437.367,176.923,16.036,152.034
C08814=1098.806,127.895,437.384,176.921,16.036,152.035
C08815=1098.801,127.681,437.401,176.919,16.036,152.035
C08816=1098.797,127.465,437.417,176.915,16.036,152.036
C08817=1098.792,127.251,437.434,176.913,16.036,152.036
C08818=1098.786,127.036,437.451,176.911,16.036,152.037
C08819=1098.781,126.820,437.469,176.908,16.036,152.037
C08820=1098.776,126.572,437.488,176.905,16.036,152.038
C08821=1098.770,126.323,437.508,176.902,16.035,152.038
C08822=1098.765,126.074,437.527,176.899,16.035,152.039
C08823=1098.759,125.825,437.547,176.896,16.035,152.040
C08824=1098.753,125.575,437.566,176.893,16.035,152.040
C08825=1098.747,125.326,437.585,176.890,16.035,152.041
C08826=1098.741,125.077,437.605,176.887,16.034,152.041
C08827=1098.736,124.827,437.625,176.884,16.034,152.042
C08828=1098.731,124.578,437.644,176.881,16.034,152.042
C08829=1098.725,124.329,437.664,176.879,16.034,152.043
C08830=1098.719,124.080,437.684,176.875,16.034,152.044
C08831=1098.714,123.831,437.702,176.872,16.033,152.044
C08832=1098.708,123.582,437.722,176.870,16.034,152.045
C08833=1098.702,123.333,437.742,176.866,16.033,152.045
C08834=1098.697,123.083,437.761,176.864,16.033,152.046
C08835=1098.691,122.834,437.781,176.861,16.033,152.046
C08836=1098.685,122.585,437.800,176.857,16.033,152.047
C08837=1098.679,122.336,437.819,176.855,16.033,152.048
C08838=1098.674,122.087,437.838,176.852,16.032,152.048
C08839=1098.668,121.838,437.858,176.849,16.032,152.049
C08840=1098.662,121.589,437.877,176.846,16.032,152.049
C08841=1098.657,121.339,437.897,176.843,16.032,152.050
C08842=1098.652,121.089,437.917,176.840,16.032,152.050
C08843=1098.646,120.840,437.936,176.837,16.031,152.051
C08844=1098.641,120.592,437.955,176.834,16.032,152.052
C08845=1098.635,120.342,437.975,176.831,16.031,152.052
C08846=1098.629,120.093,437.994,176.828,16.030,152.053
C08847=1098.624,119.844,438.013,176.826,16.030,152.053
C08848=1098.618,119.594,438.032,176.822,16.030,152.054
C08849=1098.613,119.345,438.051,176.820,16.030,152.054
C08850=1098.607,119.097,438.071,176.817,16.030,152.055
C08851=1098.601,118.847,438.090,176.813,16.029,152.055
C08852=1098.595,118.598,438.110,176.811,16.030,152.056
C08853=1098.590,118.349,438.129,176.808,16.029,152.056
C08854=1098.585,118.100,438.148,176.805,16.029,152.057
C08855=1098.579,117.850,438.167,176.802,16.029,152.058
C08856=1098.573,117.601,438.186,176.800,16.029,152.058
C08857=1098.568,117.352,438.205,176.797,16.028,152.059
C08858=1098.562,117.103,438.224,176.793,16.027,152.059
C08859=1098.556,116.853,438.243,176.791,16.028,152.060
C08860=1098.551,116.605,438.262,176.788,16.027,152.060
C08861=1098.545,116.355,438.281,176.786,16.027,152.061
C08862=1098.540,116.106,438.300,176.782,16.027,152.061
C08863=1098.534,115.856,438.320,176.779,16.026,152.062
C08864=1098.526,115.514,438.346,176.775,16.026,152.063
C08865=1098.519,115.171,438.372,176.771,16.025,152.063
C08866=1098.512,114.828,438.398,176.768,16.025,152.064
C08867=1098.504,114.486,438.424,176.763,16.025,152.065
C08868=1098.498,114.236,438.444,176.761,16.025,152.065
C08869=1098.493,113.987,438.463,176.758,16.024,152.066
C08870=1098.486,113.738,438.482,176.756,16.024,152.066
C08871=1098.481,113.489,438.500,176.752,16.024,152.067
C08872=1098.475,113.239,438.520,176.749,16.023,152.067
C08873=1098.470,112.990,438.539,176.747,16.023,152.068
C08874=1098.464,112.742,438.557,176.744,16.023,152.068
C08875=1098.459,112.491,438.576,176.741,16.023,152.069
C08876=1098.452,112.217,438.597,176.738,16.022,152.070
C08877=1098.446,111.943,438.618,176.735,16.022,152.070
C08878=1098.439,111.669,438.639,176.732,16.021,152.071
C08879=1098.434,111.395,438.659,176.728,16.021,152.071
C08880=1098.428,111.145,438.678,176.726,16.021,152.072
C08881=1098.423,110.897,438.697,176.723,16.021,152.072
C08882=1098.417,110.647,438.716,176.720,16.020,152.073
C08883=1098.411,110.398,438.734,176.717,16.020,152.073
C08884=1098.406,110.149,438.753,176.715,16.020,152.074
C08885=1098.399,109.900,438.772,176.712,16.019,152.074
C08886=1098.394,109.650,438.791,176.709,16.019,152.075
C08887=1098.388,109.401,438.810,176.706,16.019,152.076
C08888=1098.382,109.152,438.828,176.703,16.018,152.076
C08889=1098.377,108.902,438.847,176.700,16.018,152.076
C08890=1098.372,108.654,438.866,176.697,16.018,152.077
C08891=1098.366,108.404,438.884,176.695,16.018,152.077
C08892=1098.360,108.154,438.903,176.692,16.017,152.078
C08893=1098.354,107.906,438.921,176.690,16.017,152.078
C08894=1098.348,107.657,438.940,176.686,16.017,152.079
C08895=1098.343,107.407,438.959,176.684,16.016,152.079
C08896=1098.337,107.158,438.977,176.681,16.016,152.080
C08897=1098.331,106.909,438.996,176.678,16.016,152.081
C08898=1098.326,106.660,439.014,176.675,16.015,152.081
C08899=1098.320,106.410,439.033,176.672,16.015,152.082
C08900=1098.315,106.161,439.052,176.670,16.015,152.082
C08901=1098.309,105.912,439.070,176.667,16.014,152.083
C08902=1098.303,105.662,439.089,176.664,16.014,152.083
C08903=1098.298,105.413,439.107,176.661,16.014,152.084
C08904=1098.292,105.164,439.126,176.659,16.013,152.084
C08905=1098.286,104.915,439.145,176.656,16.013,152.085
C08906=1098.281,104.665,439.163,176.653,16.012,152.085
C08907=1098.275,104.416,439.182,176.650,16.012,152.086
C08908=1098.270,104.167,439.200,176.647,16.011,152.086
C08909=1098.263,103.918,439.218,176.645,16.011,152.086
C08910=1098.259,103.668,439.237,176.642,16.011,152.087
C08911=1098.253,103.419,439.256,176.640,16.010,152.087
C08912=1098.247,103.170,439.273,176.636,16.010,152.088
C08913=1098.242,102.921,439.293,176.634,16.010,152.088
C08914=1098.236,102.671,439.310,176.631,16.009,152.089
C08915=1098.230,102.422,439.329,176.629,16.009,152.089
C08916=1098.225,102.173,439.347,176.626,16.008,152.090
C08917=1098.219,101.924,439.366,176.623,16.008,152.090
C08918=1098.214,101.675,439.384,176.620,16.008,152.091
C08919=1098.208,101.425,439.403,176.617,16.007,152.091
C08920=1098.202,101.176,439.421,176.615,16.007,152.092
C08921=1098.196,100.926,439.439,176.612,16.006,152.092
C08922=1098.191,100.677,439.458,176.609,16.006,152.093
C08923=1098.185,100.428,439.475,176.607,16.005,152.093
C08924=1098.179,100.179,439.494,176.604,16.005,152.094
C08925=1098.174,99.929,439.512,176.601,16.005,152.094
C08926=1098.168,99.680,439.531,176.599,16.005,152.095
C08927=1098.162,99.431,439.548,176.596,16.004,152.095
C08928=1098.157,99.181,439.567,176.593,16.004,152.096
C08929=1098.151,98.933,439.585,176.590,16.003,152.096
C08930=1098.145,98.683,439.603,176.588,16.003,152.097
C08931=1098.140,98.434,439.621,176.585,16.002,152.097
C08932=1098.133,98.185,439.640,176.582,16.001,152.097
C08933=1098.128,97.935,439.657,176.580,16.002,152.098
C08934=1098.123,97.685,439.676,176.577,16.001,152.098
C08935=1098.117,97.437,439.694,176.574,16.001,152.099
C08936=1098.111,97.187,439.712,176.571,16.000,152.099
C08937=1098.106,96.938,439.730,176.569,16.000,152.100
C08938=1098.100,96.689,439.748,176.566,15.999,152.100
C08939=1098.094,96.440,439.767,176.564,15.999,152.101
C08940=1098.088,96.166,439.786,176.561,15.998,152.101
C08941=1098.082,95.891,439.806,176.558,15.998,152.102
C08942=1098.075,95.618,439.826,176.554,15.997,152.102
C08943=1098.069,95.343,439.846,176.552,15.997,152.103
C08944=1098.063,95.094,439.863,176.549,15.997,152.103
C08945=1098.058,94.845,439.882,176.547,15.996,152.104
C08946=1098.052,94.595,439.900,176.544,15.995,152.104
C08947=1098.047,94.346,439.918,176.542,15.995,152.104
C08948=1098.041,94.097,439.935,176.539,15.994,152.105
C08949=1098.036,93.847,439.954,176.536,15.995,152.105
C08950=1098.030,93.598,439.971,176.533,15.994,152.106
C08951=1098.024,93.349,439.990,176.531,15.993,152.106
C08952=1098.018,93.100,440.008,176.528,15.993,152.107
C08953=1098.013,92.850,440.026,176.525,15.992,152.107
C08954=1098.007,92.601,440.044,176.523,15.991,152.108
C08955=1098.002,92.352,440.061,176.519,15.991,152.108
C08956=1097.996,92.103,440.079,176.517,15.991,152.109
C08957=1097.990,91.853,440.097,176.514,15.990,152.109
C08958=1097.985,91.604,440.115,176.512,15.990,152.109
C08959=1097.979,91.354,440.133,176.509,15.989,152.110
C08960=1097.974,91.105,440.151,176.507,15.989,152.110
C08961=1097.968,90.856,440.168,176.504,15.988,152.111
C08962=1097.962,90.606,440.186,176.502,15.987,152.111
C08963=1097.956,90.358,440.204,176.499,15.987,152.112
C08964=1097.951,90.108,440.222,176.496,15.987,152.112
C08965=1097.945,89.859,440.240,176.493,15.986,152.113
C08966=1097.939,89.610,440.257,176.491,15.986,152.113
C08967=1097.933,89.360,440.275,176.488,15.985,152.113
C08968=1097.927,89.111,440.293,176.486,15.985,152.114
C08969=1097.922,88.862,440.310,176.483,15.984,152.114
C08970=1097.916,88.612,440.328,176.481,15.983,152.115
C08971=1097.910,88.363,440.346,176.478,15.983,152.115
C08972=1097.905,88.114,440.363,176.475,15.983,152.116
C08973=1097.899,87.864,440.381,176.473,15.982,152.116
C08974=1097.893,87.615,440.398,176.470,15.982,152.116
C08975=1097.888,87.366,440.416,176.467,15.981,152.117
C08976=1097.882,87.116,440.434,176.465,15.981,152.117
C08977=1097.876,86.867,440.451,176.462,15.980,152.118
C08978=1097.871,86.618,440.469,176.460,15.980,152.118
C08979=1097.865,86.368,440.487,176.457,15.979,152.119
C08980=1097.859,86.119,440.504,176.455,15.978,152.119
C08981=1097.854,85.870,440.522,176.452,15.978,152.119
C08982=1097.848,85.621,440.540,176.450,15.977,152.120
C08983=1097.842,85.371,440.557,176.447,15.976,152.120
C08984=1097.837,85.122,440.574,176.445,15.976,152.121
C08985=1097.831,84.872,440.592,176.442,15.975,152.121
C08986=1097.825,84.623,440.610,176.439,15.975,152.121
C08987=1097.820,84.374,440.627,176.436,15.974,152.122
C08988=1097.814,84.125,440.645,176.434,15.974,152.122
C08989=1097.809,83.875,440.662,176.431,15.973,152.123
C08990=1097.803,83.625,440.680,176.429,15.973,152.123
C08991=1097.797,83.376,440.697,176.426,15.972,152.124
C08992=1097.792,83.127,440.715,176.424,15.972,152.124
C08993=1097.786,82.878,440.732,176.421,15.971,152.124
C08994=1097.780,82.628,440.750,176.419,15.971,152.125
C08995=1097.775,82.379,440.767,176.417,15.970,152.125
C08996=1097.769,82.130,440.784,176.414,15.969,152.125
C08997=1097.763,81.880,440.801,176.412,15.969,152.126
C08998=1097.758,81.631,440.819,176.409,15.968,152.126
C08999=1097.752,81.382,440.837,176.407,15.968,152.127
C09000=1097.747,81.132,440.853,176.404,15.967,152.127
C09001=1097.741,80.883,440.871,176.401,15.967,152.128
C09002=1097.735,80.634,440.889,176.398,15.966,152.128
C09003=1097.730,80.385,440.906,176.397,15.965,152.128
C09004=1097.724,80.110,440.925,176.394,15.964,152.129
C09005=1097.717,79.836,440.944,176.391,15.963,152.129
C09006=1097.711,79.562,440.963,176.388,15.963,152.130
C09007=1097.705,79.288,440.982,176.385,15.962,152.130
C09008=1097.699,79.038,440.999,176.382,15.961,152.130
C09009=1097.693,78.789,441.016,176.380,15.961,152.131
C09010=1097.688,78.540,441.033,176.377,15.960,152.131
C09011=1097.682,78.291,441.051,176.375,15.960,152.132
C09012=1097.677,78.042,441.068,176.372,15.959,152.132
C09013=1097.672,77.792,441.085,176.370,15.959,152.132
C09014=1097.665,77.543,441.102,176.367,15.958,152.133
C09015=1097.660,77.293,441.119,176.365,15.957,152.133
C09016=1097.654,77.044,441.137,176.362,15.957,152.134
C09017=1097.648,76.794,441.153,176.360,15.956,152.134
C09018=1097.643,76.545,441.171,176.358,15.956,152.134
C09019=1097.637,76.296,441.187,176.355,15.955,152.135
C09020=1097.631,76.046,441.205,176.353,15.955,152.135
C09021=1097.625,75.797,441.222,176.350,15.954,152.136
C09022=1097.620,75.548,441.239,176.348,15.953,152.136
C09023=1097.614,75.298,441.255,176.345,15.952,152.136
C09024=1097.608,75.049,441.273,176.343,15.952,152.137
C09025=1097.603,74.800,441.290,176.340,15.951,152.137
C09026=1097.597,74.551,441.307,176.338,15.951,152.137
C09027=1097.591,74.301,441.324,176.335,15.950,152.138
C09028=1097.586,74.051,441.342,176.333,15.949,152.138
C09029=1097.580,73.802,441.358,176.330,15.948,152.139
C09030=1097.574,73.553,441.375,176.328,15.948,152.139
C09031=1097.569,73.303,441.392,176.325,15.947,152.139
C09032=1097.563,73.054,441.409,176.323,15.947,152.140
C09033=1097.557,72.805,441.426,176.321,15.946,152.140
C09034=1097.552,72.555,441.443,176.318,15.945,152.140
C09035=1097.546,72.307,441.460,176.316,15.945,152.141
C09036=1097.541,72.057,441.477,176.313,15.944,152.141
C09037=1097.534,71.807,441.493,176.311,15.943,152.141
C09038=1097.529,71.558,441.511,176.308,15.942,152.142
C09039=1097.523,71.308,441.528,176.306,15.942,152.142
C09040=1097.517,71.059,441.544,176.303,15.941,152.143
C09041=1097.512,70.810,441.562,176.301,15.941,152.143
C09042=1097.506,70.561,441.578,176.298,15.939,152.143
C09043=1097.501,70.311,441.595,176.296,15.939,152.144
C09044=1097.495,70.062,441.612,176.294,15.939,152.144
C09045=1097.489,69.812,441.629,176.291,15.937,152.144
C09046=1097.483,69.563,441.645,176.289,15.937,152.145
C09047=1097.478,69.314,441.662,176.286,15.936,152.145
C09048=1097.472,69.065,441.679,176.284,15.936,152.145
C09049=1097.467,68.815,441.696,176.281,15.935,152.146
C09050=1097.461,68.566,441.712,176.279,15.935,152.146
C09051=1097.455,68.317,441.729,176.276,15.933,152.147
C09052=1097.449,68.067,441.746,176.274,15.933,152.147
C09053=1097.444,67.818,441.762,176.272,15.932,152.147
C09054=1097.438,67.568,441.779,176.269,15.932,152.148
C09055=1097.433,67.319,441.796,176.267,15.931,152.148
C09056=1097.427,67.070,441.813,176.264,15.930,152.148
C09057=1097.421,66.820,441.829,176.262,15.930,152.149
C09058=1097.415,66.571,441.846,176.260,15.928,152.149
C09059=1097.410,66.321,441.863,176.257,15.928,152.149
C09060=1097.404,66.072,441.879,176.255,15.927,152.150
C09061=1097.398,65.823,441.895,176.253,15.927,152.150
C09062=1097.393,65.574,441.913,176.251,15.926,152.150
C09063=1097.387,65.324,441.929,176.248,15.925,152.151
C09064=1097.382,65.075,441.946,176.245,15.925,152.151
C09065=1097.376,64.825,441.962,176.243,15.923,152.151
C09066=1097.370,64.576,441.978,176.241,15.923,152.152
C09067=1097.365,64.326,441.995,176.238,15.922,152.152
C09068=1097.357,64.052,442.013,176.236,15.922,152.153
C09069=1097.351,63.777,442.032,176.233,15.921,152.153
C09070=1097.345,63.504,442.050,176.230,15.920,152.153
C09071=1097.338,63.230,442.068,176.228,15.919,152.154
